gfCNCPoint2[7249] = {X 509.8909, Y 46.0603, Z -3.0000, A 0.000, B 0.000, C 0.000 }
gfCNCPoint2[7250] = {X 509.6596, Y 47.0980, Z -3.0000, A 0.000, B 0.000, C 0.000 }
gfCNCPoint2[7251] = {X 509.2797, Y 48.0910, Z -3.0000, A 0.000, B 0.000, C 0.000 }
gfCNCPoint2[7252] = {X 508.7593, Y 49.0180, Z -3.0000, A 0.000, B 0.000, C 0.000 }
gfCNCPoint2[7253] = {X 508.0200, Y 49.9571, Z -3.0000, A 0.000, B 0.000, C 0.000 }
gfCNCPoint2[7254] = {X 507.1371, Y 50.7626, Z -3.0000, A 0.000, B 0.000, C 0.000 }
gfCNCPoint2[7255] = {X 506.1343, Y 51.4129, Z -3.0000, A 0.000, B 0.000, C 0.000 }
gfCNCPoint2[7256] = {X 505.0386, Y 51.8902, Z -3.0000, A 0.000, B 0.000, C 0.000 }
gfCNCPoint2[7257] = {X 503.8796, Y 52.1819, Z -3.0000, A 0.000, B 0.000, C 0.000 }
gfCNCPoint2[7258] = {X 502.6885, Y 52.2800, Z -3.0000, A 0.000, B 0.000, C 0.000 }
gfCNCPoint2[7259] = {X 496.2450, Y 52.2800, Z -3.0000, A 0.000, B 0.000, C 0.000 }
gfCNCPoint2[7260] = {X 495.0845, Y 52.1869, Z -3.0000, A 0.000, B 0.000, C 0.000 }
gfCNCPoint2[7261] = {X 493.9538, Y 51.9100, Z -3.0000, A 0.000, B 0.000, C 0.000 }
gfCNCPoint2[7262] = {X 492.8816, Y 51.4564, Z -3.0000, A 0.000, B 0.000, C 0.000 }
gfCNCPoint2[7263] = {X 491.8954, Y 50.8377, Z -3.0000, A 0.000, B 0.000, C 0.000 }
gfCNCPoint2[7264] = {X 491.0204, Y 50.0697, Z -3.0000, A 0.000, B 0.000, C 0.000 }
gfCNCPoint2[7265] = {X 490.2980, Y 49.1989, Z -3.0000, A 0.000, B 0.000, C 0.000 }
gfCNCPoint2[7266] = {X 489.7192, Y 48.2267, Z -3.0000, A 0.000, B 0.000, C 0.000 }
gfCNCPoint2[7267] = {X 489.2980, Y 47.1766, Z -3.0000, A 0.000, B 0.000, C 0.000 }
gfCNCPoint2[7268] = {X 488.8769, Y 48.2267, Z -3.0000, A 0.000, B 0.000, C 0.000 }
gfCNCPoint2[7269] = {X 488.2981, Y 49.1989, Z -3.0000, A 0.000, B 0.000, C 0.000 }
gfCNCPoint2[7270] = {X 487.5756, Y 50.0697, Z -3.0000, A 0.000, B 0.000, C 0.000 }
gfCNCPoint2[7271] = {X 486.8824, Y 50.6978, Z -3.0000, A 0.000, B 0.000, C 0.000 }
gfCNCPoint2[7272] = {X 486.1145, Y 51.2318, Z -3.0000, A 0.000, B 0.000, C 0.000 }
gfCNCPoint2[7273] = {X 485.2843, Y 51.6629, Z -3.0000, A 0.000, B 0.000, C 0.000 }
gfCNCPoint2[7274] = {X 486.0586, Y 53.1385, Z -3.0000, A 0.000, B 0.000, C 0.000 }
gfCNCPoint2[7275] = {X 486.6224, Y 54.7067, Z -3.0000, A 0.000, B 0.000, C 0.000 }
gfCNCPoint2[7276] = {X 486.9651, Y 56.3375, Z -3.0000, A 0.000, B 0.000, C 0.000 }
gfCNCPoint2[7277] = {X 487.0800, Y 58.0000, Z -3.0000, A 0.000, B 0.000, C 0.000 }
gfCNCPoint2[7278] = {X 487.0796, Y 59.0339, Z -3.0000, A 0.000, B 0.000, C 0.000 }
gfCNCPoint2[7279] = {X 486.9596, Y 60.6353, Z -3.0000, A 0.000, B 0.000, C 0.000 }
gfCNCPoint2[7280] = {X 486.6283, Y 62.2067, Z -3.0000, A 0.000, B 0.000, C 0.000 }
gfCNCPoint2[7281] = {X 486.0914, Y 63.7202, Z -3.0000, A 0.000, B 0.000, C 0.000 }
gfCNCPoint2[7282] = {X 485.3585, Y 65.1491, Z -3.0000, A 0.000, B 0.000, C 0.000 }
gfCNCPoint2[7283] = {X 484.4426, Y 66.4682, Z -3.0000, A 0.000, B 0.000, C 0.000 }
gfCNCPoint2[7284] = {X 483.3598, Y 67.6542, Z -3.0000, A 0.000, B 0.000, C 0.000 }
gfCNCPoint2[7285] = {X 483.3601, Y 88.3509, Z -3.0000, A 0.000, B 0.000, C 0.000 }
gfCNCPoint2[7286] = {X 484.3099, Y 89.3715, Z -3.0000, A 0.000, B 0.000, C 0.000 }
gfCNCPoint2[7287] = {X 485.1356, Y 90.4950, Z -3.0000, A 0.000, B 0.000, C 0.000 }
gfCNCPoint2[7288] = {X 507.6818, Y 90.4950, Z -3.0000, A 0.000, B 0.000, C 0.000 }
gfCNCPoint2[7289] = {X 507.6818, Y 92.8950, Z -3.0000, A 0.000, B 0.000, C 0.000 }
gfCNCPoint2[7290] = {X 592.8965, Y 92.8950, Z -3.0000, A 0.000, B 0.000, C 0.000 }
gfCNCPoint2[7291] = {X 592.8965, Y 56.5812, Z -3.0000, A 0.000, B 0.000, C 0.000 }
gfCNCPoint2[7292] = {X 591.4810, Y 56.4128, Z -3.0000, A 0.000, B 0.000, C 0.000 }
gfCNCPoint2[7293] = {X 590.0968, Y 56.0720, Z -3.0000, A 0.000, B 0.000, C 0.000 }
gfCNCPoint2[7294] = {X 588.7648, Y 55.5641, Z -3.0000, A 0.000, B 0.000, C 0.000 }
gfCNCPoint2[7295] = {X 587.5052, Y 54.8965, Z -3.0000, A 0.000, B 0.000, C 0.000 }
gfCNCPoint2[7296] = {X 586.9690, Y 55.2051, Z -3.0000, A 0.000, B 0.000, C 0.000 }
gfCNCPoint2[7297] = {X 586.4171, Y 55.4846, Z -3.0000, A 0.000, B 0.000, C 0.000 }
gfCNCPoint2[7298] = {X 584.8782, Y 56.0830, Z -3.0000, A 0.000, B 0.000, C 0.000 }
gfCNCPoint2[7299] = {X 583.2699, Y 56.4570, Z -3.0000, A 0.000, B 0.000, C 0.000 }
gfCNCPoint2[7300] = {X 581.6248, Y 56.5987, Z -3.0000, A 0.000, B 0.000, C 0.000 }
gfCNCPoint2[7301] = {X 579.9763, Y 56.5055, Z -3.0000, A 0.000, B 0.000, C 0.000 }
gfCNCPoint2[7302] = {X 578.3577, Y 56.1792, Z -3.0000, A 0.000, B 0.000, C 0.000 }
gfCNCPoint2[7303] = {X 576.8018, Y 55.6263, Z -3.0000, A 0.000, B 0.000, C 0.000 }
gfCNCPoint2[7304] = {X 575.3401, Y 54.8581, Z -3.0000, A 0.000, B 0.000, C 0.000 }
gfCNCPoint2[7305] = {X 573.9176, Y 55.6091, Z -3.0000, A 0.000, B 0.000, C 0.000 }
gfCNCPoint2[7306] = {X 572.4049, Y 56.1560, Z -3.0000, A 0.000, B 0.000, C 0.000 }
gfCNCPoint2[7307] = {X 570.8311, Y 56.4885, Z -3.0000, A 0.000, B 0.000, C 0.000 }
gfCNCPoint2[7308] = {X 569.2264, Y 56.6000, Z -3.0000, A 0.000, B 0.000, C 0.000 }
gfCNCPoint2[7309] = {X 562.4443, Y 56.6000, Z -3.0000, A 0.000, B 0.000, C 0.000 }
gfCNCPoint2[7310] = {X 560.8792, Y 56.4939, Z -3.0000, A 0.000, B 0.000, C 0.000 }
gfCNCPoint2[7311] = {X 559.3428, Y 56.1777, Z -3.0000, A 0.000, B 0.000, C 0.000 }
gfCNCPoint2[7312] = {X 557.8630, Y 55.6570, Z -3.0000, A 0.000, B 0.000, C 0.000 }
gfCNCPoint2[7313] = {X 556.4671, Y 54.9415, Z -3.0000, A 0.000, B 0.000, C 0.000 }
gfCNCPoint2[7314] = {X 555.1804, Y 54.0441, Z -3.0000, A 0.000, B 0.000, C 0.000 }
gfCNCPoint2[7315] = {X 554.0266, Y 52.9814, Z -3.0000, A 0.000, B 0.000, C 0.000 }
gfCNCPoint2[7316] = {X 553.0267, Y 51.7727, Z -3.0000, A 0.000, B 0.000, C 0.000 }
gfCNCPoint2[7317] = {X 552.1991, Y 50.4401, Z -3.0000, A 0.000, B 0.000, C 0.000 }
gfCNCPoint2[7318] = {X 551.5587, Y 49.0081, Z -3.0000, A 0.000, B 0.000, C 0.000 }
gfCNCPoint2[7319] = {X 551.1637, Y 47.7032, Z -3.0000, A 0.000, B 0.000, C 0.000 }
gfCNCPoint2[7320] = {X 550.9244, Y 46.3610, Z -3.0000, A 0.000, B 0.000, C 0.000 }
gfCNCPoint2[7321] = {X 550.8443, Y 45.0000, Z -3.0000, A 0.000, B 0.000, C 0.000 }
gfCNCPoint2[7322] = {X 550.8443, Y 44.0535, Z -3.0000, A 0.000, B 0.000, C 0.000 }
gfCNCPoint2[7323] = {X 550.9571, Y 42.4679, Z -3.0000, A 0.000, B 0.000, C 0.000 }
gfCNCPoint2[7324] = {X 551.2850, Y 40.9124, Z -3.0000, A 0.000, B 0.000, C 0.000 }
gfCNCPoint2[7325] = {X 551.8218, Y 39.4161, Z -3.0000, A 0.000, B 0.000, C 0.000 }
gfCNCPoint2[7326] = {X 549.6234, Y 38.4533, Z -3.0000, A 0.000, B 0.000, C 0.000 }
gfCNCPoint2[7327] = {X 549.7925, Y 38.0819, Z -3.0000, A 0.000, B 0.000, C 0.000 }
gfCNCPoint2[7328] = {X 549.9724, Y 37.7156, Z -3.0000, A 0.000, B 0.000, C 0.000 }
gfCNCPoint2[7329] = {X 549.9724, Y 16.9500, Z -3.0000, A 0.000, B 0.000, C 0.000 }
gfCNCPoint2[7330] = {X 549.8029, Y 17.1990, Z -3.0000, A 0.000, B 0.000, C 0.000 }
gfCNCPoint2[7331] = {X 549.6232, Y 17.4407, Z -3.0000, A 0.000, B 0.000, C 0.000 }
gfCNCPoint2[7332] = {X 549.6234, Y 38.4533, Z -3.0000, A 0.000, B 0.000, C 0.000 }
gfCNCPoint2[7333] = {X 551.8218, Y 39.4161, Z -3.0000, A 0.000, B 0.000, C 0.000 }
gfCNCPoint2[7334] = {X 552.0826, Y 38.8609, Z -3.0000, A 0.000, B 0.000, C 0.000 }
gfCNCPoint2[7335] = {X 552.3724, Y 38.3202, Z -3.0000, A 0.000, B 0.000, C 0.000 }
gfCNCPoint2[7336] = {X 552.3724, Y 11.6888, Z -3.0000, A 0.000, B 0.000, C 0.000 }
gfCNCPoint2[7337] = {X 551.6708, Y 10.2343, Z -3.0000, A 0.000, B 0.000, C 0.000 }
gfCNCPoint2[7338] = {X 551.1780, Y 8.6964, Z -3.0000, A 0.000, B 0.000, C 0.000 }
gfCNCPoint2[7339] = {X 550.9035, Y 7.1050, Z -3.0000, A 0.000, B 0.000, C 0.000 }
gfCNCPoint2[7340] = {X 524.2928, Y 7.1050, Z -3.0000, A 0.000, B 0.000, C 0.000 }
gfCNCPoint2[7341] = {X 524.3789, Y 7.2067, Z -3.0000, A 0.000, B 0.000, C 0.000 }
gfCNCPoint2[7342] = {X 524.4621, Y 7.3107, Z -3.0000, A 0.000, B 0.000, C 0.000 }
gfCNCPoint2[7343] = {X 543.7426, Y 7.3112, Z -3.0000, A 0.000, B 0.000, C 0.000 }
gfCNCPoint2[7344] = {X 544.7118, Y 7.3834, Z -3.0000, A 0.000, B 0.000, C 0.000 }
gfCNCPoint2[7345] = {X 545.6475, Y 7.6459, Z -3.0000, A 0.000, B 0.000, C 0.000 }
gfCNCPoint2[7346] = {X 546.5127, Y 8.0885, Z -3.0000, A 0.000, B 0.000, C 0.000 }
gfCNCPoint2[7347] = {X 547.2732, Y 8.6936, Z -3.0000, A 0.000, B 0.000, C 0.000 }
gfCNCPoint2[7348] = {X 547.8989, Y 9.4373, Z -3.0000, A 0.000, B 0.000, C 0.000 }
gfCNCPoint2[7349] = {X 548.3649, Y 10.2901, Z -3.0000, A 0.000, B 0.000, C 0.000 }
gfCNCPoint2[7350] = {X 548.6529, Y 11.2183, Z -3.0000, A 0.000, B 0.000, C 0.000 }
gfCNCPoint2[7351] = {X 548.7514, Y 12.1852, Z -3.0000, A 0.000, B 0.000, C 0.000 }
gfCNCPoint2[7352] = {X 548.7512, Y 13.0283, Z -3.0000, A 0.000, B 0.000, C 0.000 }
gfCNCPoint2[7353] = {X 548.6549, Y 13.9439, Z -3.0000, A 0.000, B 0.000, C 0.000 }
gfCNCPoint2[7354] = {X 548.3884, Y 14.8251, Z -3.0000, A 0.000, B 0.000, C 0.000 }
gfCNCPoint2[7355] = {X 547.9611, Y 15.6406, Z -3.0000, A 0.000, B 0.000, C 0.000 }
gfCNCPoint2[7356] = {X 547.6183, Y 16.1045, Z -3.0000, A 0.000, B 0.000, C 0.000 }
gfCNCPoint2[7357] = {X 547.2232, Y 16.5248, Z -3.0000, A 0.000, B 0.000, C 0.000 }
gfCNCPoint2[7358] = {X 547.2234, Y 40.6622, Z -3.0000, A 0.000, B 0.000, C 0.000 }
gfCNCPoint2[7359] = {X 547.8650, Y 41.4042, Z -3.0000, A 0.000, B 0.000, C 0.000 }
gfCNCPoint2[7360] = {X 548.3452, Y 42.2595, Z -3.0000, A 0.000, B 0.000, C 0.000 }
gfCNCPoint2[7361] = {X 548.6447, Y 43.1936, Z -3.0000, A 0.000, B 0.000, C 0.000 }
gfCNCPoint2[7362] = {X 548.7513, Y 44.1687, Z -3.0000, A 0.000, B 0.000, C 0.000 }
gfCNCPoint2[7363] = {X 548.7514, Y 45.0016, Z -3.0000, A 0.000, B 0.000, C 0.000 }
gfCNCPoint2[7364] = {X 548.6696, Y 45.8828, Z -3.0000, A 0.000, B 0.000, C 0.000 }
gfCNCPoint2[7365] = {X 548.4300, Y 46.7348, Z -3.0000, A 0.000, B 0.000, C 0.000 }
gfCNCPoint2[7366] = {X 548.0407, Y 47.5296, Z -3.0000, A 0.000, B 0.000, C 0.000 }
gfCNCPoint2[7367] = {X 547.5144, Y 48.2411, Z -3.0000, A 0.000, B 0.000, C 0.000 }
gfCNCPoint2[7368] = {X 546.7288, Y 48.9506, Z -3.0000, A 0.000, B 0.000, C 0.000 }
gfCNCPoint2[7369] = {X 545.8088, Y 49.4742, Z -3.0000, A 0.000, B 0.000, C 0.000 }
gfCNCPoint2[7370] = {X 544.7975, Y 49.7874, Z -3.0000, A 0.000, B 0.000, C 0.000 }
gfCNCPoint2[7371] = {X 543.7426, Y 49.8753, Z -3.0000, A 0.000, B 0.000, C 0.000 }
gfCNCPoint2[7372] = {X 524.3233, Y 49.8758, Z -3.0000, A 0.000, B 0.000, C 0.000 }
gfCNCPoint2[7373] = {X 523.7105, Y 50.5147, Z -3.0000, A 0.000, B 0.000, C 0.000 }
gfCNCPoint2[7374] = {X 522.9953, Y 51.0365, Z -3.0000, A 0.000, B 0.000, C 0.000 }
gfCNCPoint2[7375] = {X 522.1999, Y 51.4251, Z -3.0000, A 0.000, B 0.000, C 0.000 }
gfCNCPoint2[7376] = {X 521.3487, Y 51.6685, Z -3.0000, A 0.000, B 0.000, C 0.000 }
gfCNCPoint2[7377] = {X 520.4681, Y 51.7591, Z -3.0000, A 0.000, B 0.000, C 0.000 }
gfCNCPoint2[7378] = {X 519.7998, Y 51.7591, Z -3.0000, A 0.000, B 0.000, C 0.000 }
gfCNCPoint2[7379] = {X 518.8477, Y 51.6654, Z -3.0000, A 0.000, B 0.000, C 0.000 }
gfCNCPoint2[7380] = {X 517.9323, Y 51.3877, Z -3.0000, A 0.000, B 0.000, C 0.000 }
gfCNCPoint2[7381] = {X 517.0886, Y 50.9367, Z -3.0000, A 0.000, B 0.000, C 0.000 }
gfCNCPoint2[7382] = {X 516.3491, Y 50.3298, Z -3.0000, A 0.000, B 0.000, C 0.000 }
gfCNCPoint2[7383] = {X 515.7422, Y 49.5903, Z -3.0000, A 0.000, B 0.000, C 0.000 }
gfCNCPoint2[7384] = {X 515.2912, Y 48.7466, Z -3.0000, A 0.000, B 0.000, C 0.000 }
gfCNCPoint2[7385] = {X 515.0135, Y 47.8312, Z -3.0000, A 0.000, B 0.000, C 0.000 }
gfCNCPoint2[7386] = {X 514.9198, Y 46.8791, Z -3.0000, A 0.000, B 0.000, C 0.000 }
gfCNCPoint2[7387] = {X 514.9198, Y 39.9011, Z -3.0000, A 0.000, B 0.000, C 0.000 }
gfCNCPoint2[7388] = {X 515.0197, Y 38.9186, Z -3.0000, A 0.000, B 0.000, C 0.000 }
gfCNCPoint2[7389] = {X 515.3154, Y 37.9764, Z -3.0000, A 0.000, B 0.000, C 0.000 }
gfCNCPoint2[7390] = {X 515.7947, Y 37.1129, Z -3.0000, A 0.000, B 0.000, C 0.000 }
gfCNCPoint2[7391] = {X 516.4381, Y 36.3637, Z -3.0000, A 0.000, B 0.000, C 0.000 }
gfCNCPoint2[7392] = {X 517.2191, Y 35.7593, Z -3.0000, A 0.000, B 0.000, C 0.000 }
gfCNCPoint2[7393] = {X 518.1058, Y 35.3245, Z -3.0000, A 0.000, B 0.000, C 0.000 }
gfCNCPoint2[7394] = {X 519.0619, Y 35.0772, Z -3.0000, A 0.000, B 0.000, C 0.000 }
gfCNCPoint2[7395] = {X 519.4084, Y 35.0368, Z -3.0000, A 0.000, B 0.000, C 0.000 }
gfCNCPoint2[7396] = {X 519.7568, Y 35.0213, Z -3.0000, A 0.000, B 0.000, C 0.000 }
gfCNCPoint2[7397] = {X 520.5345, Y 35.0216, Z -3.0000, A 0.000, B 0.000, C 0.000 }
gfCNCPoint2[7398] = {X 521.4086, Y 35.1126, Z -3.0000, A 0.000, B 0.000, C 0.000 }
gfCNCPoint2[7399] = {X 522.2522, Y 35.3589, Z -3.0000, A 0.000, B 0.000, C 0.000 }
gfCNCPoint2[7400] = {X 523.0379, Y 35.7525, Z -3.0000, A 0.000, B 0.000, C 0.000 }
gfCNCPoint2[7401] = {X 523.7403, Y 36.2806, Z -3.0000, A 0.000, B 0.000, C 0.000 }
gfCNCPoint2[7402] = {X 524.3366, Y 36.9262, Z -3.0000, A 0.000, B 0.000, C 0.000 }
gfCNCPoint2[7403] = {X 534.0719, Y 36.9267, Z -3.0000, A 0.000, B 0.000, C 0.000 }
gfCNCPoint2[7404] = {X 534.0719, Y 34.5249, Z -3.0000, A 0.000, B 0.000, C 0.000 }
gfCNCPoint2[7405] = {X 530.3966, Y 34.5246, Z -3.0000, A 0.000, B 0.000, C 0.000 }
gfCNCPoint2[7406] = {X 529.7967, Y 35.1733, Z -3.0000, A 0.000, B 0.000, C 0.000 }
gfCNCPoint2[7407] = {X 529.0897, Y 35.7033, Z -3.0000, A 0.000, B 0.000, C 0.000 }
gfCNCPoint2[7408] = {X 528.2986, Y 36.0971, Z -3.0000, A 0.000, B 0.000, C 0.000 }
gfCNCPoint2[7409] = {X 527.4495, Y 36.3417, Z -3.0000, A 0.000, B 0.000, C 0.000 }
gfCNCPoint2[7410] = {X 526.5703, Y 36.4293, Z -3.0000, A 0.000, B 0.000, C 0.000 }
gfCNCPoint2[7411] = {X 525.8868, Y 36.4294, Z -3.0000, A 0.000, B 0.000, C 0.000 }
gfCNCPoint2[7412] = {X 524.9094, Y 36.3306, Z -3.0000, A 0.000, B 0.000, C 0.000 }
gfCNCPoint2[7413] = {X 523.9717, Y 36.0380, Z -3.0000, A 0.000, B 0.000, C 0.000 }
gfCNCPoint2[7414] = {X 523.1116, Y 35.5636, Z -3.0000, A 0.000, B 0.000, C 0.000 }
gfCNCPoint2[7415] = {X 522.3639, Y 34.9265, Z -3.0000, A 0.000, B 0.000, C 0.000 }
gfCNCPoint2[7416] = {X 521.7590, Y 34.1525, Z -3.0000, A 0.000, B 0.000, C 0.000 }
gfCNCPoint2[7417] = {X 521.3213, Y 33.2731, Z -3.0000, A 0.000, B 0.000, C 0.000 }
gfCNCPoint2[7418] = {X 521.0686, Y 32.3239, Z -3.0000, A 0.000, B 0.000, C 0.000 }
gfCNCPoint2[7419] = {X 521.0222, Y 31.9379, Z -3.0000, A 0.000, B 0.000, C 0.000 }
gfCNCPoint2[7420] = {X 521.0068, Y 31.5495, Z -3.0000, A 0.000, B 0.000, C 0.000 }
gfCNCPoint2[7421] = {X 521.0076, Y 24.4815, Z -3.0000, A 0.000, B 0.000, C 0.000 }
gfCNCPoint2[7422] = {X 521.0984, Y 23.6300, Z -3.0000, A 0.000, B 0.000, C 0.000 }
gfCNCPoint2[7423] = {X 521.3368, Y 22.8074, Z -3.0000, A 0.000, B 0.000, C 0.000 }
gfCNCPoint2[7424] = {X 521.7152, Y 22.0391, Z -3.0000, A 0.000, B 0.000, C 0.000 }
gfCNCPoint2[7425] = {X 521.1864, Y 22.1316, Z -3.0000, A 0.000, B 0.000, C 0.000 }
gfCNCPoint2[7426] = {X 520.6505, Y 22.1656, Z -3.0000, A 0.000, B 0.000, C 0.000 }
gfCNCPoint2[7427] = {X 519.9691, Y 22.1657, Z -3.0000, A 0.000, B 0.000, C 0.000 }
gfCNCPoint2[7428] = {X 519.5109, Y 22.1442, Z -3.0000, A 0.000, B 0.000, C 0.000 }
gfCNCPoint2[7429] = {X 519.0567, Y 22.0797, Z -3.0000, A 0.000, B 0.000, C 0.000 }
gfCNCPoint2[7430] = {X 518.1336, Y 21.8074, Z -3.0000, A 0.000, B 0.000, C 0.000 }
gfCNCPoint2[7431] = {X 517.2820, Y 21.3592, Z -3.0000, A 0.000, B 0.000, C 0.000 }
gfCNCPoint2[7432] = {X 516.5348, Y 20.7527, Z -3.0000, A 0.000, B 0.000, C 0.000 }
gfCNCPoint2[7433] = {X 515.9212, Y 20.0113, Z -3.0000, A 0.000, B 0.000, C 0.000 }
gfCNCPoint2[7434] = {X 515.4650, Y 19.1639, Z -3.0000, A 0.000, B 0.000, C 0.000 }
gfCNCPoint2[7435] = {X 515.1840, Y 18.2434, Z -3.0000, A 0.000, B 0.000, C 0.000 }
gfCNCPoint2[7436] = {X 515.0891, Y 17.2857, Z -3.0000, A 0.000, B 0.000, C 0.000 }
gfCNCPoint2[7437] = {X 515.0891, Y 10.3077, Z -3.0000, A 0.000, B 0.000, C 0.000 }
gfCNCPoint2[7438] = {X 515.0965, Y 10.0383, Z -3.0000, A 0.000, B 0.000, C 0.000 }
gfCNCPoint2[7439] = {X 515.1189, Y 9.7697, Z -3.0000, A 0.000, B 0.000, C 0.000 }
gfCNCPoint2[7440] = {X 515.3251, Y 8.8084, Z -3.0000, A 0.000, B 0.000, C 0.000 }
gfCNCPoint2[7441] = {X 515.7199, Y 7.9080, Z -3.0000, A 0.000, B 0.000, C 0.000 }
gfCNCPoint2[7442] = {X 516.2871, Y 7.1050, Z -3.0000, A 0.000, B 0.000, C 0.000 }
gfCNCPoint2[7443] = {X 516.6492, Y 7.4201, Z -3.0000, A 0.000, B 0.000, C 0.000 }
gfCNCPoint2[7444] = {X 517.3373, Y 6.7816, Z -3.0000, A 0.000, B 0.000, C 0.000 }
gfCNCPoint2[7445] = {X 518.1451, Y 6.3036, Z -3.0000, A 0.000, B 0.000, C 0.000 }
gfCNCPoint2[7446] = {X 519.0359, Y 6.0078, Z -3.0000, A 0.000, B 0.000, C 0.000 }
gfCNCPoint2[7447] = {X 519.9692, Y 5.9077, Z -3.0000, A 0.000, B 0.000, C 0.000 }
gfCNCPoint2[7448] = {X 520.6509, Y 5.9079, Z -3.0000, A 0.000, B 0.000, C 0.000 }
gfCNCPoint2[7449] = {X 521.4834, Y 5.9951, Z -3.0000, A 0.000, B 0.000, C 0.000 }
gfCNCPoint2[7450] = {X 522.2844, Y 6.2384, Z -3.0000, A 0.000, B 0.000, C 0.000 }
gfCNCPoint2[7451] = {X 523.0248, Y 6.6290, Z -3.0000, A 0.000, B 0.000, C 0.000 }
gfCNCPoint2[7452] = {X 523.6778, Y 7.1528, Z -3.0000, A 0.000, B 0.000, C 0.000 }
gfCNCPoint2[7453] = {X 524.2198, Y 7.7907, Z -3.0000, A 0.000, B 0.000, C 0.000 }
gfCNCPoint2[7454] = {X 543.7489, Y 7.7912, Z -3.0000, A 0.000, B 0.000, C 0.000 }
gfCNCPoint2[7455] = {X 544.7470, Y 7.8786, Z -3.0000, A 0.000, B 0.000, C 0.000 }
gfCNCPoint2[7456] = {X 545.6995, Y 8.1892, Z -3.0000, A 0.000, B 0.000, C 0.000 }
gfCNCPoint2[7457] = {X 546.5572, Y 8.7070, Z -3.0000, A 0.000, B 0.000, C 0.000 }
gfCNCPoint2[7458] = {X 547.2757, Y 9.4052, Z -3.0000, A 0.000, B 0.000, C 0.000 }
gfCNCPoint2[7459] = {X 547.8178, Y 10.2477, Z -3.0000, A 0.000, B 0.000, C 0.000 }
gfCNCPoint2[7460] = {X 548.1556, Y 11.1909, Z -3.0000, A 0.000, B 0.000, C 0.000 }
gfCNCPoint2[7461] = {X 548.2714, Y 12.1861, Z -3.0000, A 0.000, B 0.000, C 0.000 }
gfCNCPoint2[7462] = {X 548.2712, Y 13.0233, Z -3.0000, A 0.000, B 0.000, C 0.000 }
gfCNCPoint2[7463] = {X 548.1628, Y 13.9496, Z -3.0000, A 0.000, B 0.000, C 0.000 }
gfCNCPoint2[7464] = {X 547.8617, Y 14.8322, Z -3.0000, A 0.000, B 0.000, C 0.000 }
gfCNCPoint2[7465] = {X 547.3813, Y 15.6315, Z -3.0000, A 0.000, B 0.000, C 0.000 }
gfCNCPoint2[7466] = {X 546.7432, Y 16.3116, Z -3.0000, A 0.000, B 0.000, C 0.000 }
gfCNCPoint2[7467] = {X 546.7434, Y 40.8754, Z -3.0000, A 0.000, B 0.000, C 0.000 }
gfCNCPoint2[7468] = {X 547.3883, Y 41.5646, Z -3.0000, A 0.000, B 0.000, C 0.000 }
gfCNCPoint2[7469] = {X 547.8713, Y 42.3754, Z -3.0000, A 0.000, B 0.000, C 0.000 }
gfCNCPoint2[7470] = {X 548.1702, Y 43.2706, Z -3.0000, A 0.000, B 0.000, C 0.000 }
gfCNCPoint2[7471] = {X 548.2714, Y 44.2089, Z -3.0000, A 0.000, B 0.000, C 0.000 }
gfCNCPoint2[7472] = {X 548.2714, Y 45.0007, Z -3.0000, A 0.000, B 0.000, C 0.000 }
gfCNCPoint2[7473] = {X 548.1556, Y 45.9959, Z -3.0000, A 0.000, B 0.000, C 0.000 }
gfCNCPoint2[7474] = {X 547.8178, Y 46.9391, Z -3.0000, A 0.000, B 0.000, C 0.000 }
gfCNCPoint2[7475] = {X 547.2757, Y 47.7816, Z -3.0000, A 0.000, B 0.000, C 0.000 }
gfCNCPoint2[7476] = {X 546.5572, Y 48.4798, Z -3.0000, A 0.000, B 0.000, C 0.000 }
gfCNCPoint2[7477] = {X 545.6995, Y 48.9975, Z -3.0000, A 0.000, B 0.000, C 0.000 }
gfCNCPoint2[7478] = {X 544.7469, Y 49.3080, Z -3.0000, A 0.000, B 0.000, C 0.000 }
gfCNCPoint2[7479] = {X 543.7489, Y 49.3953, Z -3.0000, A 0.000, B 0.000, C 0.000 }
gfCNCPoint2[7480] = {X 524.0859, Y 49.3958, Z -3.0000, A 0.000, B 0.000, C 0.000 }
gfCNCPoint2[7481] = {X 523.5292, Y 50.0308, Z -3.0000, A 0.000, B 0.000, C 0.000 }
gfCNCPoint2[7482] = {X 522.8649, Y 50.5523, Z -3.0000, A 0.000, B 0.000, C 0.000 }
gfCNCPoint2[7483] = {X 522.1158, Y 50.9422, Z -3.0000, A 0.000, B 0.000, C 0.000 }
gfCNCPoint2[7484] = {X 521.3076, Y 51.1873, Z -3.0000, A 0.000, B 0.000, C 0.000 }
gfCNCPoint2[7485] = {X 520.4681, Y 51.2791, Z -3.0000, A 0.000, B 0.000, C 0.000 }
gfCNCPoint2[7486] = {X 519.7998, Y 51.2791, Z -3.0000, A 0.000, B 0.000, C 0.000 }
gfCNCPoint2[7487] = {X 518.8207, Y 51.1688, Z -3.0000, A 0.000, B 0.000, C 0.000 }
gfCNCPoint2[7488] = {X 517.8907, Y 50.8434, Z -3.0000, A 0.000, B 0.000, C 0.000 }
gfCNCPoint2[7489] = {X 517.0564, Y 50.3192, Z -3.0000, A 0.000, B 0.000, C 0.000 }
gfCNCPoint2[7490] = {X 516.3597, Y 49.6225, Z -3.0000, A 0.000, B 0.000, C 0.000 }
gfCNCPoint2[7491] = {X 515.8355, Y 48.7882, Z -3.0000, A 0.000, B 0.000, C 0.000 }
gfCNCPoint2[7492] = {X 515.5101, Y 47.8582, Z -3.0000, A 0.000, B 0.000, C 0.000 }
gfCNCPoint2[7493] = {X 515.3998, Y 46.8791, Z -3.0000, A 0.000, B 0.000, C 0.000 }
gfCNCPoint2[7494] = {X 515.3998, Y 39.9011, Z -3.0000, A 0.000, B 0.000, C 0.000 }
gfCNCPoint2[7495] = {X 515.5101, Y 38.9220, Z -3.0000, A 0.000, B 0.000, C 0.000 }
gfCNCPoint2[7496] = {X 515.8355, Y 37.9920, Z -3.0000, A 0.000, B 0.000, C 0.000 }
gfCNCPoint2[7497] = {X 516.3597, Y 37.1577, Z -3.0000, A 0.000, B 0.000, C 0.000 }
gfCNCPoint2[7498] = {X 517.0565, Y 36.4610, Z -3.0000, A 0.000, B 0.000, C 0.000 }
gfCNCPoint2[7499] = {X 517.8907, Y 35.9368, Z -3.0000, A 0.000, B 0.000, C 0.000 }
gfCNCPoint2[7500] = {X 518.8207, Y 35.6114, Z -3.0000, A 0.000, B 0.000, C 0.000 }
gfCNCPoint2[7501] = {X 519.7999, Y 35.5011, Z -3.0000, A 0.000, B 0.000, C 0.000 }
gfCNCPoint2[7502] = {X 520.5280, Y 35.5015, Z -3.0000, A 0.000, B 0.000, C 0.000 }
gfCNCPoint2[7503] = {X 521.3615, Y 35.5927, Z -3.0000, A 0.000, B 0.000, C 0.000 }
gfCNCPoint2[7504] = {X 522.1626, Y 35.8404, Z -3.0000, A 0.000, B 0.000, C 0.000 }
gfCNCPoint2[7505] = {X 522.9022, Y 36.2356, Z -3.0000, A 0.000, B 0.000, C 0.000 }
gfCNCPoint2[7506] = {X 523.5534, Y 36.7640, Z -3.0000, A 0.000, B 0.000, C 0.000 }
gfCNCPoint2[7507] = {X 524.0925, Y 37.4062, Z -3.0000, A 0.000, B 0.000, C 0.000 }
gfCNCPoint2[7508] = {X 534.5519, Y 37.4067, Z -3.0000, A 0.000, B 0.000, C 0.000 }
gfCNCPoint2[7509] = {X 534.5519, Y 34.0450, Z -3.0000, A 0.000, B 0.000, C 0.000 }
gfCNCPoint2[7510] = {X 530.1526, Y 34.0445, Z -3.0000, A 0.000, B 0.000, C 0.000 }
gfCNCPoint2[7511] = {X 529.6049, Y 34.6951, Z -3.0000, A 0.000, B 0.000, C 0.000 }
gfCNCPoint2[7512] = {X 528.9423, Y 35.2282, Z -3.0000, A 0.000, B 0.000, C 0.000 }
gfCNCPoint2[7513] = {X 528.1895, Y 35.6238, Z -3.0000, A 0.000, B 0.000, C 0.000 }
gfCNCPoint2[7514] = {X 527.3747, Y 35.8673, Z -3.0000, A 0.000, B 0.000, C 0.000 }
gfCNCPoint2[7515] = {X 526.5283, Y 35.9495, Z -3.0000, A 0.000, B 0.000, C 0.000 }
gfCNCPoint2[7516] = {X 525.8868, Y 35.9495, Z -3.0000, A 0.000, B 0.000, C 0.000 }
gfCNCPoint2[7517] = {X 524.9077, Y 35.8391, Z -3.0000, A 0.000, B 0.000, C 0.000 }
gfCNCPoint2[7518] = {X 523.9777, Y 35.5137, Z -3.0000, A 0.000, B 0.000, C 0.000 }
gfCNCPoint2[7519] = {X 523.1434, Y 34.9895, Z -3.0000, A 0.000, B 0.000, C 0.000 }
gfCNCPoint2[7520] = {X 522.4467, Y 34.2928, Z -3.0000, A 0.000, B 0.000, C 0.000 }
gfCNCPoint2[7521] = {X 521.9225, Y 33.4585, Z -3.0000, A 0.000, B 0.000, C 0.000 }
gfCNCPoint2[7522] = {X 521.5971, Y 32.5285, Z -3.0000, A 0.000, B 0.000, C 0.000 }
gfCNCPoint2[7523] = {X 521.4868, Y 31.5495, Z -3.0000, A 0.000, B 0.000, C 0.000 }
gfCNCPoint2[7524] = {X 521.4868, Y 24.5714, Z -3.0000, A 0.000, B 0.000, C 0.000 }
gfCNCPoint2[7525] = {X 521.5971, Y 23.5923, Z -3.0000, A 0.000, B 0.000, C 0.000 }
gfCNCPoint2[7526] = {X 521.9225, Y 22.6623, Z -3.0000, A 0.000, B 0.000, C 0.000 }
gfCNCPoint2[7527] = {X 522.4467, Y 21.8281, Z -3.0000, A 0.000, B 0.000, C 0.000 }
gfCNCPoint2[7528] = {X 523.1434, Y 21.1314, Z -3.0000, A 0.000, B 0.000, C 0.000 }
gfCNCPoint2[7529] = {X 523.9777, Y 20.6072, Z -3.0000, A 0.000, B 0.000, C 0.000 }
gfCNCPoint2[7530] = {X 524.9077, Y 20.2817, Z -3.0000, A 0.000, B 0.000, C 0.000 }
gfCNCPoint2[7531] = {X 525.8868, Y 20.1714, Z -3.0000, A 0.000, B 0.000, C 0.000 }
gfCNCPoint2[7532] = {X 526.5702, Y 20.1716, Z -3.0000, A 0.000, B 0.000, C 0.000 }
gfCNCPoint2[7533] = {X 527.4024, Y 20.2591, Z -3.0000, A 0.000, B 0.000, C 0.000 }
gfCNCPoint2[7534] = {X 528.2030, Y 20.5025, Z -3.0000, A 0.000, B 0.000, C 0.000 }
gfCNCPoint2[7535] = {X 528.9430, Y 20.8931, Z -3.0000, A 0.000, B 0.000, C 0.000 }
gfCNCPoint2[7536] = {X 529.5956, Y 21.4167, Z -3.0000, A 0.000, B 0.000, C 0.000 }
gfCNCPoint2[7537] = {X 530.1374, Y 22.0544, Z -3.0000, A 0.000, B 0.000, C 0.000 }
gfCNCPoint2[7538] = {X 534.5519, Y 22.0547, Z -3.0000, A 0.000, B 0.000, C 0.000 }
gfCNCPoint2[7539] = {X 534.5519, Y 19.7814, Z -3.0000, A 0.000, B 0.000, C 0.000 }
gfCNCPoint2[7540] = {X 528.8167, Y 19.7812, Z -3.0000, A 0.000, B 0.000, C 0.000 }
gfCNCPoint2[7541] = {X 528.8167, Y 20.2612, Z -3.0000, A 0.000, B 0.000, C 0.000 }
gfCNCPoint2[7542] = {X 534.0719, Y 20.2614, Z -3.0000, A 0.000, B 0.000, C 0.000 }
gfCNCPoint2[7543] = {X 534.0719, Y 21.5747, Z -3.0000, A 0.000, B 0.000, C 0.000 }
gfCNCPoint2[7544] = {X 530.3797, Y 21.5744, Z -3.0000, A 0.000, B 0.000, C 0.000 }
gfCNCPoint2[7545] = {X 529.6676, Y 20.8352, Z -3.0000, A 0.000, B 0.000, C 0.000 }
gfCNCPoint2[7546] = {X 528.8167, Y 20.2612, Z -3.0000, A 0.000, B 0.000, C 0.000 }
gfCNCPoint2[7547] = {X 528.8167, Y 19.7812, Z -3.0000, A 0.000, B 0.000, C 0.000 }
gfCNCPoint2[7548] = {X 524.2348, Y 19.7810, Z -3.0000, A 0.000, B 0.000, C 0.000 }
gfCNCPoint2[7549] = {X 523.6871, Y 20.4315, Z -3.0000, A 0.000, B 0.000, C 0.000 }
gfCNCPoint2[7550] = {X 523.0246, Y 20.9645, Z -3.0000, A 0.000, B 0.000, C 0.000 }
gfCNCPoint2[7551] = {X 522.2718, Y 21.3601, Z -3.0000, A 0.000, B 0.000, C 0.000 }
gfCNCPoint2[7552] = {X 521.4571, Y 21.6036, Z -3.0000, A 0.000, B 0.000, C 0.000 }
gfCNCPoint2[7553] = {X 520.6107, Y 21.6857, Z -3.0000, A 0.000, B 0.000, C 0.000 }
gfCNCPoint2[7554] = {X 519.9691, Y 21.6857, Z -3.0000, A 0.000, B 0.000, C 0.000 }
gfCNCPoint2[7555] = {X 518.9900, Y 21.5754, Z -3.0000, A 0.000, B 0.000, C 0.000 }
gfCNCPoint2[7556] = {X 518.0600, Y 21.2500, Z -3.0000, A 0.000, B 0.000, C 0.000 }
gfCNCPoint2[7557] = {X 517.2257, Y 20.7258, Z -3.0000, A 0.000, B 0.000, C 0.000 }
gfCNCPoint2[7558] = {X 516.5290, Y 20.0291, Z -3.0000, A 0.000, B 0.000, C 0.000 }
gfCNCPoint2[7559] = {X 516.0048, Y 19.1948, Z -3.0000, A 0.000, B 0.000, C 0.000 }
gfCNCPoint2[7560] = {X 515.6794, Y 18.2648, Z -3.0000, A 0.000, B 0.000, C 0.000 }
gfCNCPoint2[7561] = {X 515.5691, Y 17.2857, Z -3.0000, A 0.000, B 0.000, C 0.000 }
gfCNCPoint2[7562] = {X 515.5691, Y 10.3077, Z -3.0000, A 0.000, B 0.000, C 0.000 }
gfCNCPoint2[7563] = {X 515.6394, Y 9.5244, Z -3.0000, A 0.000, B 0.000, C 0.000 }
gfCNCPoint2[7564] = {X 515.8480, Y 8.7662, Z -3.0000, A 0.000, B 0.000, C 0.000 }
gfCNCPoint2[7565] = {X 516.1882, Y 8.0572, Z -3.0000, A 0.000, B 0.000, C 0.000 }
gfCNCPoint2[7566] = {X 516.6492, Y 7.4201, Z -3.0000, A 0.000, B 0.000, C 0.000 }
gfCNCPoint2[7567] = {X 516.2871, Y 7.1050, Z -3.0000, A 0.000, B 0.000, C 0.000 }
gfCNCPoint2[7568] = {X 469.2610, Y 7.1050, Z -3.0000, A 0.000, B 0.000, C 0.000 }
gfCNCPoint2[7569] = {X 469.2610, Y 11.9050, Z -3.0000, A 0.000, B 0.000, C 0.000 }
gfCNCPoint2[7570] = {X 469.1140, Y 11.9050, Z -3.0000, A 0.000, B 0.000, C 0.000 }
gfCNCPoint2[7571] = {X 469.1169, Y 12.0441, Z -3.0000, A 0.000, B 0.000, C 0.000 }
gfCNCPoint2[7572] = {X 469.1179, Y 12.1832, Z -3.0000, A 0.000, B 0.000, C 0.000 }
gfCNCPoint2[7573] = {X 469.1888, Y 12.0438, Z -3.0000, A 0.000, B 0.000, C 0.000 }
gfCNCPoint2[7574] = {X 469.2610, Y 11.9050, Z -3.0000, A 0.000, B 0.000, C 0.000 }
gfCNCPoint2[7575] = {X 469.2610, Y 9.5050, Z -3.0000, A 0.000, B 0.000, C 0.000 }
gfCNCPoint2[7576] = {X 466.2070, Y 9.5050, Z -3.0000, A 0.000, B 0.000, C 0.000 }
gfCNCPoint2[7577] = {X 466.5688, Y 10.7173, Z -3.0000, A 0.000, B 0.000, C 0.000 }
gfCNCPoint2[7578] = {X 466.7149, Y 11.9739, Z -3.0000, A 0.000, B 0.000, C 0.000 }
gfCNCPoint2[7579] = {X 466.7172, Y 12.0782, Z -3.0000, A 0.000, B 0.000, C 0.000 }
gfCNCPoint2[7580] = {X 466.7179, Y 12.1826, Z -3.0000, A 0.000, B 0.000, C 0.000 }
gfCNCPoint2[7581] = {X 466.7179, Y 12.9779, Z -3.0000, A 0.000, B 0.000, C 0.000 }
gfCNCPoint2[7582] = {X 466.6191, Y 14.1736, Z -3.0000, A 0.000, B 0.000, C 0.000 }
gfCNCPoint2[7583] = {X 466.3252, Y 15.3368, Z -3.0000, A 0.000, B 0.000, C 0.000 }
gfCNCPoint2[7584] = {X 465.8443, Y 16.4359, Z -3.0000, A 0.000, B 0.000, C 0.000 }
gfCNCPoint2[7585] = {X 465.1893, Y 17.4412, Z -3.0000, A 0.000, B 0.000, C 0.000 }
gfCNCPoint2[7586] = {X 465.1897, Y 25.8716, Z -3.0000, A 0.000, B 0.000, C 0.000 }
gfCNCPoint2[7587] = {X 467.5897, Y 25.8714, Z -3.0000, A 0.000, B 0.000, C 0.000 }
gfCNCPoint2[7588] = {X 467.5904, Y 38.9895, Z -3.0000, A 0.000, B 0.000, C 0.000 }
gfCNCPoint2[7589] = {X 467.6015, Y 39.0069, Z -3.0000, A 0.000, B 0.000, C 0.000 }
gfCNCPoint2[7590] = {X 468.3506, Y 37.9855, Z -3.0000, A 0.000, B 0.000, C 0.000 }
gfCNCPoint2[7591] = {X 469.2267, Y 37.0706, Z -3.0000, A 0.000, B 0.000, C 0.000 }
gfCNCPoint2[7592] = {X 470.2148, Y 36.2780, Z -3.0000, A 0.000, B 0.000, C 0.000 }
gfCNCPoint2[7593] = {X 471.5280, Y 33.7075, Z -3.0000, A 0.000, B 0.000, C 0.000 }
gfCNCPoint2[7594] = {X 470.4811, Y 32.4115, Z -3.0000, A 0.000, B 0.000, C 0.000 }
gfCNCPoint2[7595] = {X 469.5675, Y 31.0183, Z -3.0000, A 0.000, B 0.000, C 0.000 }
gfCNCPoint2[7596] = {X 468.7961, Y 29.5416, Z -3.0000, A 0.000, B 0.000, C 0.000 }
gfCNCPoint2[7597] = {X 468.1745, Y 27.9959, Z -3.0000, A 0.000, B 0.000, C 0.000 }
gfCNCPoint2[7598] = {X 467.7088, Y 26.3963, Z -3.0000, A 0.000, B 0.000, C 0.000 }
gfCNCPoint2[7599] = {X 467.6476, Y 26.1342, Z -3.0000, A 0.000, B 0.000, C 0.000 }
gfCNCPoint2[7600] = {X 467.5897, Y 25.8714, Z -3.0000, A 0.000, B 0.000, C 0.000 }
gfCNCPoint2[7601] = {X 465.1897, Y 25.8716, Z -3.0000, A 0.000, B 0.000, C 0.000 }
gfCNCPoint2[7602] = {X 465.1904, Y 39.7470, Z -3.0000, A 0.000, B 0.000, C 0.000 }
gfCNCPoint2[7603] = {X 465.3903, Y 40.0173, Z -3.0000, A 0.000, B 0.000, C 0.000 }
gfCNCPoint2[7604] = {X 465.5774, Y 40.2966, Z -3.0000, A 0.000, B 0.000, C 0.000 }
gfCNCPoint2[7605] = {X 466.0634, Y 41.1919, Z -3.0000, A 0.000, B 0.000, C 0.000 }
gfCNCPoint2[7606] = {X 466.4196, Y 42.1462, Z -3.0000, A 0.000, B 0.000, C 0.000 }
gfCNCPoint2[7607] = {X 466.6392, Y 43.1408, Z -3.0000, A 0.000, B 0.000, C 0.000 }
gfCNCPoint2[7608] = {X 466.7178, Y 44.1564, Z -3.0000, A 0.000, B 0.000, C 0.000 }
gfCNCPoint2[7609] = {X 466.7179, Y 45.0000, Z -3.0000, A 0.000, B 0.000, C 0.000 }
gfCNCPoint2[7610] = {X 466.7033, Y 45.4609, Z -3.0000, A 0.000, B 0.000, C 0.000 }
gfCNCPoint2[7611] = {X 466.6596, Y 45.9200, Z -3.0000, A 0.000, B 0.000, C 0.000 }
gfCNCPoint2[7612] = {X 468.5433, Y 45.9200, Z -3.0000, A 0.000, B 0.000, C 0.000 }
gfCNCPoint2[7613] = {X 468.4996, Y 45.4609, Z -3.0000, A 0.000, B 0.000, C 0.000 }
gfCNCPoint2[7614] = {X 468.4850, Y 45.0000, Z -3.0000, A 0.000, B 0.000, C 0.000 }
gfCNCPoint2[7615] = {X 468.4850, Y 44.2090, Z -3.0000, A 0.000, B 0.000, C 0.000 }
gfCNCPoint2[7616] = {X 468.5580, Y 43.1798, Z -3.0000, A 0.000, B 0.000, C 0.000 }
gfCNCPoint2[7617] = {X 468.7759, Y 42.1714, Z -3.0000, A 0.000, B 0.000, C 0.000 }
gfCNCPoint2[7618] = {X 469.1341, Y 41.2038, Z -3.0000, A 0.000, B 0.000, C 0.000 }
gfCNCPoint2[7619] = {X 469.6255, Y 40.2966, Z -3.0000, A 0.000, B 0.000, C 0.000 }
gfCNCPoint2[7620] = {X 470.3102, Y 39.3876, Z -3.0000, A 0.000, B 0.000, C 0.000 }
gfCNCPoint2[7621] = {X 471.1282, Y 38.5964, Z -3.0000, A 0.000, B 0.000, C 0.000 }
gfCNCPoint2[7622] = {X 472.0595, Y 37.9424, Z -3.0000, A 0.000, B 0.000, C 0.000 }
gfCNCPoint2[7623] = {X 474.4571, Y 33.2493, Z -3.0000, A 0.000, B 0.000, C 0.000 }
gfCNCPoint2[7624] = {X 473.2258, Y 32.0046, Z -3.0000, A 0.000, B 0.000, C 0.000 }
gfCNCPoint2[7625] = {X 472.1543, Y 30.6200, Z -3.0000, A 0.000, B 0.000, C 0.000 }
gfCNCPoint2[7626] = {X 471.2583, Y 29.1158, Z -3.0000, A 0.000, B 0.000, C 0.000 }
gfCNCPoint2[7627] = {X 470.5511, Y 27.5141, Z -3.0000, A 0.000, B 0.000, C 0.000 }
gfCNCPoint2[7628] = {X 470.0431, Y 25.8386, Z -3.0000, A 0.000, B 0.000, C 0.000 }
gfCNCPoint2[7629] = {X 469.9884, Y 25.6042, Z -3.0000, A 0.000, B 0.000, C 0.000 }
gfCNCPoint2[7630] = {X 469.9366, Y 25.3692, Z -3.0000, A 0.000, B 0.000, C 0.000 }
gfCNCPoint2[7631] = {X 469.6270, Y 23.4764, Z -3.0000, A 0.000, B 0.000, C 0.000 }
gfCNCPoint2[7632] = {X 469.5028, Y 21.5625, Z -3.0000, A 0.000, B 0.000, C 0.000 }
gfCNCPoint2[7633] = {X 469.5652, Y 19.6455, Z -3.0000, A 0.000, B 0.000, C 0.000 }
gfCNCPoint2[7634] = {X 469.8136, Y 17.7437, Z -3.0000, A 0.000, B 0.000, C 0.000 }
gfCNCPoint2[7635] = {X 470.2458, Y 15.8751, Z -3.0000, A 0.000, B 0.000, C 0.000 }
gfCNCPoint2[7636] = {X 470.6919, Y 14.5440, Z -3.0000, A 0.000, B 0.000, C 0.000 }
gfCNCPoint2[7637] = {X 471.2622, Y 13.2612, Z -3.0000, A 0.000, B 0.000, C 0.000 }
gfCNCPoint2[7638] = {X 471.3232, Y 13.1413, Z -3.0000, A 0.000, B 0.000, C 0.000 }
gfCNCPoint2[7639] = {X 471.3853, Y 13.0219, Z -3.0000, A 0.000, B 0.000, C 0.000 }
gfCNCPoint2[7640] = {X 472.1263, Y 11.7667, Z -3.0000, A 0.000, B 0.000, C 0.000 }
gfCNCPoint2[7641] = {X 472.9873, Y 10.5907, Z -3.0000, A 0.000, B 0.000, C 0.000 }
gfCNCPoint2[7642] = {X 473.9599, Y 9.5050, Z -3.0000, A 0.000, B 0.000, C 0.000 }
gfCNCPoint2[7643] = {X 469.2610, Y 9.5050, Z -3.0000, A 0.000, B 0.000, C 0.000 }
gfCNCPoint2[7644] = {X 469.2610, Y 7.1050, Z -3.0000, A 0.000, B 0.000, C 0.000 }
gfCNCPoint2[7645] = {X 370.1021, Y 7.1050, Z -3.0000, A 0.000, B 0.000, C 0.000 }
gfCNCPoint2[7646] = {X 371.1257, Y 8.7920, Z -3.0000, A 0.000, B 0.000, C 0.000 }
gfCNCPoint2[7647] = {X 372.0365, Y 10.5424, Z -3.0000, A 0.000, B 0.000, C 0.000 }
gfCNCPoint2[7648] = {X 372.9307, Y 12.6018, Z -3.0000, A 0.000, B 0.000, C 0.000 }
gfCNCPoint2[7649] = {X 373.6688, Y 14.7222, Z -3.0000, A 0.000, B 0.000, C 0.000 }
gfCNCPoint2[7650] = {X 374.2467, Y 16.8917, Z -3.0000, A 0.000, B 0.000, C 0.000 }
gfCNCPoint2[7651] = {X 374.7337, Y 19.4559, Z -3.0000, A 0.000, B 0.000, C 0.000 }
gfCNCPoint2[7652] = {X 375.0386, Y 22.0481, Z -3.0000, A 0.000, B 0.000, C 0.000 }
gfCNCPoint2[7653] = {X 375.1600, Y 24.6553, Z -3.0000, A 0.000, B 0.000, C 0.000 }
gfCNCPoint2[7654] = {X 375.0972, Y 27.2646, Z -3.0000, A 0.000, B 0.000, C 0.000 }
gfCNCPoint2[7655] = {X 374.8505, Y 29.8630, Z -3.0000, A 0.000, B 0.000, C 0.000 }
gfCNCPoint2[7656] = {X 374.4212, Y 32.4374, Z -3.0000, A 0.000, B 0.000, C 0.000 }
gfCNCPoint2[7657] = {X 373.7833, Y 34.9993, Z -3.0000, A 0.000, B 0.000, C 0.000 }
gfCNCPoint2[7658] = {X 372.9218, Y 37.4948, Z -3.0000, A 0.000, B 0.000, C 0.000 }
gfCNCPoint2[7659] = {X 371.8434, Y 39.9045, Z -3.0000, A 0.000, B 0.000, C 0.000 }
gfCNCPoint2[7660] = {X 370.5564, Y 42.2096, Z -3.0000, A 0.000, B 0.000, C 0.000 }
gfCNCPoint2[7661] = {X 369.0710, Y 44.3921, Z -3.0000, A 0.000, B 0.000, C 0.000 }
gfCNCPoint2[7662] = {X 369.0323, Y 44.4442, Z -3.0000, A 0.000, B 0.000, C 0.000 }
gfCNCPoint2[7663] = {X 368.9934, Y 44.4962, Z -3.0000, A 0.000, B 0.000, C 0.000 }
gfCNCPoint2[7664] = {X 367.4735, Y 46.3510, Z -3.0000, A 0.000, B 0.000, C 0.000 }
gfCNCPoint2[7665] = {X 365.7979, Y 48.0666, Z -3.0000, A 0.000, B 0.000, C 0.000 }
gfCNCPoint2[7666] = {X 363.9795, Y 49.6299, Z -3.0000, A 0.000, B 0.000, C 0.000 }
gfCNCPoint2[7667] = {X 362.0320, Y 51.0291, Z -3.0000, A 0.000, B 0.000, C 0.000 }
gfCNCPoint2[7668] = {X 359.9702, Y 52.2536, Z -3.0000, A 0.000, B 0.000, C 0.000 }
gfCNCPoint2[7669] = {X 359.3969, Y 52.5411, Z -3.0000, A 0.000, B 0.000, C 0.000 }
gfCNCPoint2[7670] = {X 358.8172, Y 52.8153, Z -3.0000, A 0.000, B 0.000, C 0.000 }
gfCNCPoint2[7671] = {X 356.4597, Y 53.7705, Z -3.0000, A 0.000, B 0.000, C 0.000 }
gfCNCPoint2[7672] = {X 354.0251, Y 54.5078, Z -3.0000, A 0.000, B 0.000, C 0.000 }
gfCNCPoint2[7673] = {X 351.5337, Y 55.0210, Z -3.0000, A 0.000, B 0.000, C 0.000 }
gfCNCPoint2[7674] = {X 349.0060, Y 55.3059, Z -3.0000, A 0.000, B 0.000, C 0.000 }
gfCNCPoint2[7675] = {X 349.9669, Y 69.6738, Z -3.0000, A 0.000, B 0.000, C 0.000 }
gfCNCPoint2[7676] = {X 348.6528, Y 69.7412, Z -3.0000, A 0.000, B 0.000, C 0.000 }
gfCNCPoint2[7677] = {X 347.3372, Y 69.7678, Z -3.0000, A 0.000, B 0.000, C 0.000 }
gfCNCPoint2[7678] = {X 346.5719, Y 69.7765, Z -3.0000, A 0.000, B 0.000, C 0.000 }
gfCNCPoint2[7679] = {X 345.8065, Y 69.7717, Z -3.0000, A 0.000, B 0.000, C 0.000 }
gfCNCPoint2[7680] = {X 345.5896, Y 70.1915, Z -3.0000, A 0.000, B 0.000, C 0.000 }
gfCNCPoint2[7681] = {X 345.3645, Y 70.6070, Z -3.0000, A 0.000, B 0.000, C 0.000 }
gfCNCPoint2[7682] = {X 346.5773, Y 70.6173, Z -3.0000, A 0.000, B 0.000, C 0.000 }
gfCNCPoint2[7683] = {X 347.7901, Y 70.6133, Z -3.0000, A 0.000, B 0.000, C 0.000 }
gfCNCPoint2[7684] = {X 349.1241, Y 70.6191, Z -3.0000, A 0.000, B 0.000, C 0.000 }
gfCNCPoint2[7685] = {X 350.4580, Y 70.6075, Z -3.0000, A 0.000, B 0.000, C 0.000 }
gfCNCPoint2[7686] = {X 350.2073, Y 70.1433, Z -3.0000, A 0.000, B 0.000, C 0.000 }
gfCNCPoint2[7687] = {X 349.9669, Y 69.6738, Z -3.0000, A 0.000, B 0.000, C 0.000 }
gfCNCPoint2[7688] = {X 349.8068, Y 67.2792, Z -3.0000, A 0.000, B 0.000, C 0.000 }
gfCNCPoint2[7689] = {X 348.5578, Y 67.3431, Z -3.0000, A 0.000, B 0.000, C 0.000 }
gfCNCPoint2[7690] = {X 347.3074, Y 67.3679, Z -3.0000, A 0.000, B 0.000, C 0.000 }
gfCNCPoint2[7691] = {X 345.8015, Y 67.3714, Z -3.0000, A 0.000, B 0.000, C 0.000 }
gfCNCPoint2[7692] = {X 344.2965, Y 67.3197, Z -3.0000, A 0.000, B 0.000, C 0.000 }
gfCNCPoint2[7693] = {X 343.8099, Y 68.3954, Z -3.0000, A 0.000, B 0.000, C 0.000 }
gfCNCPoint2[7694] = {X 343.2656, Y 69.4431, Z -3.0000, A 0.000, B 0.000, C 0.000 }
gfCNCPoint2[7695] = {X 342.7864, Y 70.2643, Z -3.0000, A 0.000, B 0.000, C 0.000 }
gfCNCPoint2[7696] = {X 342.2717, Y 71.0638, Z -3.0000, A 0.000, B 0.000, C 0.000 }
gfCNCPoint2[7697] = {X 342.2718, Y 72.9179, Z -3.0000, A 0.000, B 0.000, C 0.000 }
gfCNCPoint2[7698] = {X 343.8005, Y 72.9735, Z -3.0000, A 0.000, B 0.000, C 0.000 }
gfCNCPoint2[7699] = {X 345.3298, Y 73.0068, Z -3.0000, A 0.000, B 0.000, C 0.000 }
gfCNCPoint2[7700] = {X 346.5590, Y 73.0173, Z -3.0000, A 0.000, B 0.000, C 0.000 }
gfCNCPoint2[7701] = {X 347.7882, Y 73.0134, Z -3.0000, A 0.000, B 0.000, C 0.000 }
gfCNCPoint2[7702] = {X 349.1414, Y 73.0190, Z -3.0000, A 0.000, B 0.000, C 0.000 }
gfCNCPoint2[7703] = {X 350.4945, Y 73.0072, Z -3.0000, A 0.000, B 0.000, C 0.000 }
gfCNCPoint2[7704] = {X 352.0276, Y 72.9726, Z -3.0000, A 0.000, B 0.000, C 0.000 }
gfCNCPoint2[7705] = {X 353.5599, Y 72.9155, Z -3.0000, A 0.000, B 0.000, C 0.000 }
gfCNCPoint2[7706] = {X 353.5598, Y 71.0781, Z -3.0000, A 0.000, B 0.000, C 0.000 }
gfCNCPoint2[7707] = {X 353.0404, Y 70.2721, Z -3.0000, A 0.000, B 0.000, C 0.000 }
gfCNCPoint2[7708] = {X 352.5571, Y 69.4440, Z -3.0000, A 0.000, B 0.000, C 0.000 }
gfCNCPoint2[7709] = {X 351.9696, Y 68.3059, Z -3.0000, A 0.000, B 0.000, C 0.000 }
gfCNCPoint2[7710] = {X 351.4503, Y 67.1351, Z -3.0000, A 0.000, B 0.000, C 0.000 }
gfCNCPoint2[7711] = {X 350.6293, Y 67.2156, Z -3.0000, A 0.000, B 0.000, C 0.000 }
gfCNCPoint2[7712] = {X 349.8068, Y 67.2792, Z -3.0000, A 0.000, B 0.000, C 0.000 }
gfCNCPoint2[7713] = {X 349.6466, Y 64.8845, Z -3.0000, A 0.000, B 0.000, C 0.000 }
gfCNCPoint2[7714] = {X 348.4628, Y 64.9450, Z -3.0000, A 0.000, B 0.000, C 0.000 }
gfCNCPoint2[7715] = {X 347.2776, Y 64.9680, Z -3.0000, A 0.000, B 0.000, C 0.000 }
gfCNCPoint2[7716] = {X 344.9731, Y 64.9481, Z -3.0000, A 0.000, B 0.000, C 0.000 }
gfCNCPoint2[7717] = {X 342.6737, Y 64.7912, Z -3.0000, A 0.000, B 0.000, C 0.000 }
gfCNCPoint2[7718] = {X 341.9389, Y 66.7262, Z -3.0000, A 0.000, B 0.000, C 0.000 }
gfCNCPoint2[7719] = {X 341.0013, Y 68.5715, Z -3.0000, A 0.000, B 0.000, C 0.000 }
gfCNCPoint2[7720] = {X 339.8716, Y 70.3059, Z -3.0000, A 0.000, B 0.000, C 0.000 }
gfCNCPoint2[7721] = {X 339.8720, Y 75.1907, Z -3.0000, A 0.000, B 0.000, C 0.000 }
gfCNCPoint2[7722] = {X 343.8270, Y 75.3752, Z -3.0000, A 0.000, B 0.000, C 0.000 }
gfCNCPoint2[7723] = {X 347.7862, Y 75.4135, Z -3.0000, A 0.000, B 0.000, C 0.000 }
gfCNCPoint2[7724] = {X 351.8753, Y 75.3780, Z -3.0000, A 0.000, B 0.000, C 0.000 }
gfCNCPoint2[7725] = {X 355.9601, Y 75.1861, Z -3.0000, A 0.000, B 0.000, C 0.000 }
gfCNCPoint2[7726] = {X 355.9597, Y 70.3191, Z -3.0000, A 0.000, B 0.000, C 0.000 }
gfCNCPoint2[7727] = {X 355.0521, Y 68.9616, Z -3.0000, A 0.000, B 0.000, C 0.000 }
gfCNCPoint2[7728] = {X 354.2626, Y 67.5321, Z -3.0000, A 0.000, B 0.000, C 0.000 }
gfCNCPoint2[7729] = {X 353.5970, Y 66.0410, Z -3.0000, A 0.000, B 0.000, C 0.000 }
gfCNCPoint2[7730] = {X 353.0598, Y 64.4989, Z -3.0000, A 0.000, B 0.000, C 0.000 }
gfCNCPoint2[7731] = {X 351.3576, Y 64.7307, Z -3.0000, A 0.000, B 0.000, C 0.000 }
gfCNCPoint2[7732] = {X 349.6466, Y 64.8845, Z -3.0000, A 0.000, B 0.000, C 0.000 }
gfCNCPoint2[7733] = {X 349.4864, Y 62.4899, Z -3.0000, A 0.000, B 0.000, C 0.000 }
gfCNCPoint2[7734] = {X 348.3678, Y 62.5468, Z -3.0000, A 0.000, B 0.000, C 0.000 }
gfCNCPoint2[7735] = {X 347.2479, Y 62.5681, Z -3.0000, A 0.000, B 0.000, C 0.000 }
gfCNCPoint2[7736] = {X 345.1177, Y 62.5519, Z -3.0000, A 0.000, B 0.000, C 0.000 }
gfCNCPoint2[7737] = {X 342.9921, Y 62.4109, Z -3.0000, A 0.000, B 0.000, C 0.000 }
gfCNCPoint2[7738] = {X 340.8784, Y 62.1457, Z -3.0000, A 0.000, B 0.000, C 0.000 }
gfCNCPoint2[7739] = {X 340.4885, Y 63.7336, Z -3.0000, A 0.000, B 0.000, C 0.000 }
gfCNCPoint2[7740] = {X 339.9471, Y 65.2766, Z -3.0000, A 0.000, B 0.000, C 0.000 }
gfCNCPoint2[7741] = {X 339.2593, Y 66.7600, Z -3.0000, A 0.000, B 0.000, C 0.000 }
gfCNCPoint2[7742] = {X 338.4316, Y 68.1701, Z -3.0000, A 0.000, B 0.000, C 0.000 }
gfCNCPoint2[7743] = {X 337.4715, Y 69.4938, Z -3.0000, A 0.000, B 0.000, C 0.000 }
gfCNCPoint2[7744] = {X 337.4721, Y 77.4162, Z -3.0000, A 0.000, B 0.000, C 0.000 }
gfCNCPoint2[7745] = {X 340.9048, Y 77.6567, Z -3.0000, A 0.000, B 0.000, C 0.000 }
gfCNCPoint2[7746] = {X 344.3433, Y 77.7892, Z -3.0000, A 0.000, B 0.000, C 0.000 }
gfCNCPoint2[7747] = {X 347.7843, Y 77.8136, Z -3.0000, A 0.000, B 0.000, C 0.000 }
gfCNCPoint2[7748] = {X 351.3134, Y 77.7927, Z -3.0000, A 0.000, B 0.000, C 0.000 }
gfCNCPoint2[7749] = {X 354.8399, Y 77.6580, Z -3.0000, A 0.000, B 0.000, C 0.000 }
gfCNCPoint2[7750] = {X 358.3603, Y 77.4095, Z -3.0000, A 0.000, B 0.000, C 0.000 }
gfCNCPoint2[7751] = {X 358.3596, Y 69.5056, Z -3.0000, A 0.000, B 0.000, C 0.000 }
gfCNCPoint2[7752] = {X 357.3486, Y 68.1061, Z -3.0000, A 0.000, B 0.000, C 0.000 }
gfCNCPoint2[7753] = {X 356.4858, Y 66.6105, Z -3.0000, A 0.000, B 0.000, C 0.000 }
gfCNCPoint2[7754] = {X 355.7802, Y 65.0347, Z -3.0000, A 0.000, B 0.000, C 0.000 }
gfCNCPoint2[7755] = {X 355.2394, Y 63.3950, Z -3.0000, A 0.000, B 0.000, C 0.000 }
gfCNCPoint2[7756] = {X 354.8689, Y 61.7086, Z -3.0000, A 0.000, B 0.000, C 0.000 }
gfCNCPoint2[7757] = {X 352.1928, Y 62.2034, Z -3.0000, A 0.000, B 0.000, C 0.000 }
gfCNCPoint2[7758] = {X 349.4864, Y 62.4899, Z -3.0000, A 0.000, B 0.000, C 0.000 }
gfCNCPoint2[7759] = {X 349.3263, Y 60.0952, Z -3.0000, A 0.000, B 0.000, C 0.000 }
gfCNCPoint2[7760] = {X 348.2728, Y 60.1487, Z -3.0000, A 0.000, B 0.000, C 0.000 }
gfCNCPoint2[7761] = {X 347.2182, Y 60.1682, Z -3.0000, A 0.000, B 0.000, C 0.000 }
gfCNCPoint2[7762] = {X 344.3864, Y 60.1133, Z -3.0000, A 0.000, B 0.000, C 0.000 }
gfCNCPoint2[7763] = {X 341.5690, Y 59.8226, Z -3.0000, A 0.000, B 0.000, C 0.000 }
gfCNCPoint2[7764] = {X 338.7856, Y 59.2982, Z -3.0000, A 0.000, B 0.000, C 0.000 }
gfCNCPoint2[7765] = {X 338.6399, Y 60.9976, Z -3.0000, A 0.000, B 0.000, C 0.000 }
gfCNCPoint2[7766] = {X 338.2959, Y 62.6682, Z -3.0000, A 0.000, B 0.000, C 0.000 }
gfCNCPoint2[7767] = {X 337.7584, Y 64.2869, Z -3.0000, A 0.000, B 0.000, C 0.000 }
gfCNCPoint2[7768] = {X 337.0347, Y 65.8314, Z -3.0000, A 0.000, B 0.000, C 0.000 }
gfCNCPoint2[7769] = {X 336.1350, Y 67.2804, Z -3.0000, A 0.000, B 0.000, C 0.000 }
gfCNCPoint2[7770] = {X 335.0715, Y 68.6139, Z -3.0000, A 0.000, B 0.000, C 0.000 }
gfCNCPoint2[7771] = {X 335.0723, Y 79.5887, Z -3.0000, A 0.000, B 0.000, C 0.000 }
gfCNCPoint2[7772] = {X 335.6732, Y 79.6587, Z -3.0000, A 0.000, B 0.000, C 0.000 }
gfCNCPoint2[7773] = {X 336.2753, Y 79.7178, Z -3.0000, A 0.000, B 0.000, C 0.000 }
gfCNCPoint2[7774] = {X 340.1046, Y 80.0147, Z -3.0000, A 0.000, B 0.000, C 0.000 }
gfCNCPoint2[7775] = {X 343.9418, Y 80.1801, Z -3.0000, A 0.000, B 0.000, C 0.000 }
gfCNCPoint2[7776] = {X 347.7824, Y 80.2137, Z -3.0000, A 0.000, B 0.000, C 0.000 }
gfCNCPoint2[7777] = {X 351.8377, Y 80.1807, Z -3.0000, A 0.000, B 0.000, C 0.000 }
gfCNCPoint2[7778] = {X 355.8892, Y 80.0006, Z -3.0000, A 0.000, B 0.000, C 0.000 }
gfCNCPoint2[7779] = {X 359.9315, Y 79.6736, Z -3.0000, A 0.000, B 0.000, C 0.000 }
gfCNCPoint2[7780] = {X 360.3463, Y 79.6320, Z -3.0000, A 0.000, B 0.000, C 0.000 }
gfCNCPoint2[7781] = {X 360.7604, Y 79.5843, Z -3.0000, A 0.000, B 0.000, C 0.000 }
gfCNCPoint2[7782] = {X 360.7596, Y 68.6242, Z -3.0000, A 0.000, B 0.000, C 0.000 }
gfCNCPoint2[7783] = {X 359.7304, Y 67.3420, Z -3.0000, A 0.000, B 0.000, C 0.000 }
gfCNCPoint2[7784] = {X 358.8533, Y 65.9514, Z -3.0000, A 0.000, B 0.000, C 0.000 }
gfCNCPoint2[7785] = {X 358.1395, Y 64.4704, Z -3.0000, A 0.000, B 0.000, C 0.000 }
gfCNCPoint2[7786] = {X 357.5981, Y 62.9179, Z -3.0000, A 0.000, B 0.000, C 0.000 }
gfCNCPoint2[7787] = {X 357.2362, Y 61.3142, Z -3.0000, A 0.000, B 0.000, C 0.000 }
gfCNCPoint2[7788] = {X 357.0917, Y 60.1647, Z -3.0000, A 0.000, B 0.000, C 0.000 }
gfCNCPoint2[7789] = {X 357.0395, Y 59.0073, Z -3.0000, A 0.000, B 0.000, C 0.000 }
gfCNCPoint2[7790] = {X 357.0394, Y 58.6377, Z -3.0000, A 0.000, B 0.000, C 0.000 }
gfCNCPoint2[7791] = {X 355.6983, Y 59.0312, Z -3.0000, A 0.000, B 0.000, C 0.000 }
gfCNCPoint2[7792] = {X 354.3416, Y 59.3673, Z -3.0000, A 0.000, B 0.000, C 0.000 }
gfCNCPoint2[7793] = {X 351.8480, Y 59.8283, Z -3.0000, A 0.000, B 0.000, C 0.000 }
gfCNCPoint2[7794] = {X 349.3263, Y 60.0952, Z -3.0000, A 0.000, B 0.000, C 0.000 }
gfCNCPoint2[7795] = {X 349.1661, Y 57.7006, Z -3.0000, A 0.000, B 0.000, C 0.000 }
gfCNCPoint2[7796] = {X 348.1779, Y 57.7505, Z -3.0000, A 0.000, B 0.000, C 0.000 }
gfCNCPoint2[7797] = {X 347.1885, Y 57.7683, Z -3.0000, A 0.000, B 0.000, C 0.000 }
gfCNCPoint2[7798] = {X 344.5488, Y 57.7187, Z -3.0000, A 0.000, B 0.000, C 0.000 }
gfCNCPoint2[7799] = {X 341.9225, Y 57.4487, Z -3.0000, A 0.000, B 0.000, C 0.000 }
gfCNCPoint2[7800] = {X 339.3279, Y 56.9602, Z -3.0000, A 0.000, B 0.000, C 0.000 }
gfCNCPoint2[7801] = {X 337.7708, Y 56.5570, Z -3.0000, A 0.000, B 0.000, C 0.000 }
gfCNCPoint2[7802] = {X 336.2363, Y 56.0750, Z -3.0000, A 0.000, B 0.000, C 0.000 }
gfCNCPoint2[7803] = {X 336.3520, Y 57.0344, Z -3.0000, A 0.000, B 0.000, C 0.000 }
gfCNCPoint2[7804] = {X 336.3907, Y 58.0000, Z -3.0000, A 0.000, B 0.000, C 0.000 }
gfCNCPoint2[7805] = {X 336.3907, Y 58.9493, Z -3.0000, A 0.000, B 0.000, C 0.000 }
gfCNCPoint2[7806] = {X 336.3894, Y 59.0917, Z -3.0000, A 0.000, B 0.000, C 0.000 }
gfCNCPoint2[7807] = {X 336.3864, Y 59.2340, Z -3.0000, A 0.000, B 0.000, C 0.000 }
gfCNCPoint2[7808] = {X 336.2427, Y 60.7983, Z -3.0000, A 0.000, B 0.000, C 0.000 }
gfCNCPoint2[7809] = {X 335.8979, Y 62.3308, Z -3.0000, A 0.000, B 0.000, C 0.000 }
gfCNCPoint2[7810] = {X 335.3577, Y 63.8059, Z -3.0000, A 0.000, B 0.000, C 0.000 }
gfCNCPoint2[7811] = {X 334.6313, Y 65.1988, Z -3.0000, A 0.000, B 0.000, C 0.000 }
gfCNCPoint2[7812] = {X 333.7308, Y 66.4859, Z -3.0000, A 0.000, B 0.000, C 0.000 }
gfCNCPoint2[7813] = {X 332.6714, Y 67.6458, Z -3.0000, A 0.000, B 0.000, C 0.000 }
gfCNCPoint2[7814] = {X 332.6725, Y 81.6423, Z -3.0000, A 0.000, B 0.000, C 0.000 }
gfCNCPoint2[7815] = {X 334.3584, Y 81.9154, Z -3.0000, A 0.000, B 0.000, C 0.000 }
gfCNCPoint2[7816] = {X 336.0555, Y 82.1077, Z -3.0000, A 0.000, B 0.000, C 0.000 }
gfCNCPoint2[7817] = {X 339.9573, Y 82.4102, Z -3.0000, A 0.000, B 0.000, C 0.000 }
gfCNCPoint2[7818] = {X 343.8671, Y 82.5790, Z -3.0000, A 0.000, B 0.000, C 0.000 }
gfCNCPoint2[7819] = {X 347.7804, Y 82.6138, Z -3.0000, A 0.000, B 0.000, C 0.000 }
gfCNCPoint2[7820] = {X 351.9132, Y 82.5796, Z -3.0000, A 0.000, B 0.000, C 0.000 }
gfCNCPoint2[7821] = {X 356.0420, Y 82.3958, Z -3.0000, A 0.000, B 0.000, C 0.000 }
gfCNCPoint2[7822] = {X 360.1614, Y 82.0626, Z -3.0000, A 0.000, B 0.000, C 0.000 }
gfCNCPoint2[7823] = {X 361.6662, Y 81.8850, Z -3.0000, A 0.000, B 0.000, C 0.000 }
gfCNCPoint2[7824] = {X 363.1606, Y 81.6342, Z -3.0000, A 0.000, B 0.000, C 0.000 }
gfCNCPoint2[7825] = {X 363.1595, Y 67.6542, Z -3.0000, A 0.000, B 0.000, C 0.000 }
gfCNCPoint2[7826] = {X 362.0732, Y 66.4639, Z -3.0000, A 0.000, B 0.000, C 0.000 }
gfCNCPoint2[7827] = {X 361.1550, Y 65.1396, Z -3.0000, A 0.000, B 0.000, C 0.000 }
gfCNCPoint2[7828] = {X 360.4213, Y 63.7049, Z -3.0000, A 0.000, B 0.000, C 0.000 }
gfCNCPoint2[7829] = {X 359.8850, Y 62.1852, Z -3.0000, A 0.000, B 0.000, C 0.000 }
gfCNCPoint2[7830] = {X 359.5558, Y 60.6078, Z -3.0000, A 0.000, B 0.000, C 0.000 }
gfCNCPoint2[7831] = {X 359.4395, Y 59.0005, Z -3.0000, A 0.000, B 0.000, C 0.000 }
gfCNCPoint2[7832] = {X 359.4393, Y 58.0000, Z -3.0000, A 0.000, B 0.000, C 0.000 }
gfCNCPoint2[7833] = {X 359.5345, Y 56.4863, Z -3.0000, A 0.000, B 0.000, C 0.000 }
gfCNCPoint2[7834] = {X 359.8187, Y 54.9964, Z -3.0000, A 0.000, B 0.000, C 0.000 }
gfCNCPoint2[7835] = {X 358.0876, Y 55.7273, Z -3.0000, A 0.000, B 0.000, C 0.000 }
gfCNCPoint2[7836] = {X 356.3147, Y 56.3497, Z -3.0000, A 0.000, B 0.000, C 0.000 }
gfCNCPoint2[7837] = {X 353.9704, Y 56.9903, Z -3.0000, A 0.000, B 0.000, C 0.000 }
gfCNCPoint2[7838] = {X 351.5825, Y 57.4416, Z -3.0000, A 0.000, B 0.000, C 0.000 }
gfCNCPoint2[7839] = {X 349.1661, Y 57.7006, Z -3.0000, A 0.000, B 0.000, C 0.000 }
gfCNCPoint2[7840] = {X 349.0060, Y 55.3059, Z -3.0000, A 0.000, B 0.000, C 0.000 }
gfCNCPoint2[7841] = {X 348.0829, Y 55.3524, Z -3.0000, A 0.000, B 0.000, C 0.000 }
gfCNCPoint2[7842] = {X 347.1589, Y 55.3683, Z -3.0000, A 0.000, B 0.000, C 0.000 }
gfCNCPoint2[7843] = {X 344.5805, Y 55.3160, Z -3.0000, A 0.000, B 0.000, C 0.000 }
gfCNCPoint2[7844] = {X 342.0169, Y 55.0362, Z -3.0000, A 0.000, B 0.000, C 0.000 }
gfCNCPoint2[7845] = {X 339.4880, Y 54.5310, Z -3.0000, A 0.000, B 0.000, C 0.000 }
gfCNCPoint2[7846] = {X 337.0137, Y 53.8044, Z -3.0000, A 0.000, B 0.000, C 0.000 }
gfCNCPoint2[7847] = {X 334.7573, Y 52.9257, Z -3.0000, A 0.000, B 0.000, C 0.000 }
gfCNCPoint2[7848] = {X 332.5817, Y 51.8629, Z -3.0000, A 0.000, B 0.000, C 0.000 }
gfCNCPoint2[7849] = {X 331.5843, Y 51.2764, Z -3.0000, A 0.000, B 0.000, C 0.000 }
gfCNCPoint2[7850] = {X 330.6109, Y 50.6508, Z -3.0000, A 0.000, B 0.000, C 0.000 }
gfCNCPoint2[7851] = {X 331.5774, Y 51.6049, Z -3.0000, A 0.000, B 0.000, C 0.000 }
gfCNCPoint2[7852] = {X 332.4009, Y 52.6848, Z -3.0000, A 0.000, B 0.000, C 0.000 }
gfCNCPoint2[7853] = {X 333.0651, Y 53.8694, Z -3.0000, A 0.000, B 0.000, C 0.000 }
gfCNCPoint2[7854] = {X 333.5571, Y 55.1352, Z -3.0000, A 0.000, B 0.000, C 0.000 }
gfCNCPoint2[7855] = {X 333.8670, Y 56.4574, Z -3.0000, A 0.000, B 0.000, C 0.000 }
gfCNCPoint2[7856] = {X 333.9597, Y 57.2262, Z -3.0000, A 0.000, B 0.000, C 0.000 }
gfCNCPoint2[7857] = {X 333.9907, Y 58.0000, Z -3.0000, A 0.000, B 0.000, C 0.000 }
gfCNCPoint2[7858] = {X 333.9907, Y 58.9450, Z -3.0000, A 0.000, B 0.000, C 0.000 }
gfCNCPoint2[7859] = {X 333.8758, Y 60.4000, Z -3.0000, A 0.000, B 0.000, C 0.000 }
gfCNCPoint2[7860] = {X 333.5444, Y 61.8214, Z -3.0000, A 0.000, B 0.000, C 0.000 }
gfCNCPoint2[7861] = {X 333.0039, Y 63.1771, Z -3.0000, A 0.000, B 0.000, C 0.000 }
gfCNCPoint2[7862] = {X 332.2664, Y 64.4366, Z -3.0000, A 0.000, B 0.000, C 0.000 }
gfCNCPoint2[7863] = {X 331.3487, Y 65.5715, Z -3.0000, A 0.000, B 0.000, C 0.000 }
gfCNCPoint2[7864] = {X 330.2713, Y 66.5561, Z -3.0000, A 0.000, B 0.000, C 0.000 }
gfCNCPoint2[7865] = {X 330.2726, Y 83.2031, Z -3.0000, A 0.000, B 0.000, C 0.000 }
gfCNCPoint2[7866] = {X 330.2763, Y 83.5834, Z -3.0000, A 0.000, B 0.000, C 0.000 }
gfCNCPoint2[7867] = {X 330.3821, Y 83.6086, Z -3.0000, A 0.000, B 0.000, C 0.000 }
gfCNCPoint2[7868] = {X 333.0927, Y 84.1520, Z -3.0000, A 0.000, B 0.000, C 0.000 }
gfCNCPoint2[7869] = {X 335.8356, Y 84.4976, Z -3.0000, A 0.000, B 0.000, C 0.000 }
gfCNCPoint2[7870] = {X 339.8099, Y 84.8057, Z -3.0000, A 0.000, B 0.000, C 0.000 }
gfCNCPoint2[7871] = {X 343.7924, Y 84.9778, Z -3.0000, A 0.000, B 0.000, C 0.000 }
gfCNCPoint2[7872] = {X 347.7785, Y 85.0139, Z -3.0000, A 0.000, B 0.000, C 0.000 }
gfCNCPoint2[7873] = {X 351.9887, Y 84.9784, Z -3.0000, A 0.000, B 0.000, C 0.000 }
gfCNCPoint2[7874] = {X 356.1948, Y 84.7909, Z -3.0000, A 0.000, B 0.000, C 0.000 }
gfCNCPoint2[7875] = {X 360.3914, Y 84.4516, Z -3.0000, A 0.000, B 0.000, C 0.000 }
gfCNCPoint2[7876] = {X 362.9937, Y 84.1047, Z -3.0000, A 0.000, B 0.000, C 0.000 }
gfCNCPoint2[7877] = {X 365.5607, Y 83.5546, Z -3.0000, A 0.000, B 0.000, C 0.000 }
gfCNCPoint2[7878] = {X 365.5594, Y 66.5618, Z -3.0000, A 0.000, B 0.000, C 0.000 }
gfCNCPoint2[7879] = {X 364.4848, Y 65.5838, Z -3.0000, A 0.000, B 0.000, C 0.000 }
gfCNCPoint2[7880] = {X 363.5688, Y 64.4560, Z -3.0000, A 0.000, B 0.000, C 0.000 }
gfCNCPoint2[7881] = {X 362.8318, Y 63.2038, Z -3.0000, A 0.000, B 0.000, C 0.000 }
gfCNCPoint2[7882] = {X 362.2906, Y 61.8554, Z -3.0000, A 0.000, B 0.000, C 0.000 }
gfCNCPoint2[7883] = {X 361.9573, Y 60.4412, Z -3.0000, A 0.000, B 0.000, C 0.000 }
gfCNCPoint2[7884] = {X 361.8395, Y 58.9930, Z -3.0000, A 0.000, B 0.000, C 0.000 }
gfCNCPoint2[7885] = {X 361.8393, Y 58.0000, Z -3.0000, A 0.000, B 0.000, C 0.000 }
gfCNCPoint2[7886] = {X 361.9156, Y 56.7870, Z -3.0000, A 0.000, B 0.000, C 0.000 }
gfCNCPoint2[7887] = {X 362.1433, Y 55.5931, Z -3.0000, A 0.000, B 0.000, C 0.000 }
gfCNCPoint2[7888] = {X 362.5747, Y 54.2990, Z -3.0000, A 0.000, B 0.000, C 0.000 }
gfCNCPoint2[7889] = {X 363.1838, Y 53.0783, Z -3.0000, A 0.000, B 0.000, C 0.000 }
gfCNCPoint2[7890] = {X 363.9585, Y 51.9554, Z -3.0000, A 0.000, B 0.000, C 0.000 }
gfCNCPoint2[7891] = {X 364.8833, Y 50.9526, Z -3.0000, A 0.000, B 0.000, C 0.000 }
gfCNCPoint2[7892] = {X 365.9399, Y 50.0897, Z -3.0000, A 0.000, B 0.000, C 0.000 }
gfCNCPoint2[7893] = {X 367.1073, Y 49.3839, Z -3.0000, A 0.000, B 0.000, C 0.000 }
gfCNCPoint2[7894] = {X 368.3624, Y 48.8492, Z -3.0000, A 0.000, B 0.000, C 0.000 }
gfCNCPoint2[7895] = {X 369.6801, Y 48.4963, Z -3.0000, A 0.000, B 0.000, C 0.000 }
gfCNCPoint2[7896] = {X 371.0344, Y 48.3322, Z -3.0000, A 0.000, B 0.000, C 0.000 }
gfCNCPoint2[7897] = {X 371.2768, Y 48.3230, Z -3.0000, A 0.000, B 0.000, C 0.000 }
gfCNCPoint2[7898] = {X 371.5193, Y 48.3200, Z -3.0000, A 0.000, B 0.000, C 0.000 }
gfCNCPoint2[7899] = {X 388.0597, Y 48.3200, Z -3.0000, A 0.000, B 0.000, C 0.000 }
gfCNCPoint2[7900] = {X 389.4419, Y 48.4192, Z -3.0000, A 0.000, B 0.000, C 0.000 }
gfCNCPoint2[7901] = {X 390.7958, Y 48.7147, Z -3.0000, A 0.000, B 0.000, C 0.000 }
gfCNCPoint2[7902] = {X 392.0936, Y 49.2006, Z -3.0000, A 0.000, B 0.000, C 0.000 }
gfCNCPoint2[7903] = {X 393.3087, Y 49.8667, Z -3.0000, A 0.000, B 0.000, C 0.000 }
gfCNCPoint2[7904] = {X 394.5333, Y 49.1962, Z -3.0000, A 0.000, B 0.000, C 0.000 }
gfCNCPoint2[7905] = {X 395.8416, Y 48.7089, Z -3.0000, A 0.000, B 0.000, C 0.000 }
gfCNCPoint2[7906] = {X 397.1858, Y 48.4177, Z -3.0000, A 0.000, B 0.000, C 0.000 }
gfCNCPoint2[7907] = {X 398.5577, Y 48.3200, Z -3.0000, A 0.000, B 0.000, C 0.000 }
gfCNCPoint2[7908] = {X 398.7346, Y 48.3200, Z -3.0000, A 0.000, B 0.000, C 0.000 }
gfCNCPoint2[7909] = {X 398.1859, Y 47.6069, Z -3.0000, A 0.000, B 0.000, C 0.000 }
gfCNCPoint2[7910] = {X 397.7774, Y 46.8051, Z -3.0000, A 0.000, B 0.000, C 0.000 }
gfCNCPoint2[7911] = {X 397.5230, Y 45.9420, Z -3.0000, A 0.000, B 0.000, C 0.000 }
gfCNCPoint2[7912] = {X 397.4561, Y 45.4921, Z -3.0000, A 0.000, B 0.000, C 0.000 }
gfCNCPoint2[7913] = {X 397.4314, Y 45.0378, Z -3.0000, A 0.000, B 0.000, C 0.000 }
gfCNCPoint2[7914] = {X 397.4316, Y 44.1456, Z -3.0000, A 0.000, B 0.000, C 0.000 }
gfCNCPoint2[7915] = {X 397.5413, Y 43.1780, Z -3.0000, A 0.000, B 0.000, C 0.000 }
gfCNCPoint2[7916] = {X 397.8410, Y 42.2514, Z -3.0000, A 0.000, B 0.000, C 0.000 }
gfCNCPoint2[7917] = {X 398.3186, Y 41.4029, Z -3.0000, A 0.000, B 0.000, C 0.000 }
gfCNCPoint2[7918] = {X 398.9552, Y 40.6660, Z -3.0000, A 0.000, B 0.000, C 0.000 }
gfCNCPoint2[7919] = {X 398.9552, Y 31.8223, Z -3.0000, A 0.000, B 0.000, C 0.000 }
gfCNCPoint2[7920] = {X 396.7484, Y 27.9866, Z -3.0000, A 0.000, B 0.000, C 0.000 }
gfCNCPoint2[7921] = {X 386.3470, Y 33.9707, Z -3.0000, A 0.000, B 0.000, C 0.000 }
gfCNCPoint2[7922] = {X 386.2661, Y 34.3977, Z -3.0000, A 0.000, B 0.000, C 0.000 }
gfCNCPoint2[7923] = {X 386.1815, Y 34.8239, Z -3.0000, A 0.000, B 0.000, C 0.000 }
gfCNCPoint2[7924] = {X 386.0225, Y 35.5735, Z -3.0000, A 0.000, B 0.000, C 0.000 }
gfCNCPoint2[7925] = {X 385.8497, Y 36.3200, Z -3.0000, A 0.000, B 0.000, C 0.000 }
gfCNCPoint2[7926] = {X 386.9552, Y 36.3200, Z -3.0000, A 0.000, B 0.000, C 0.000 }
gfCNCPoint2[7927] = {X 386.9552, Y 35.0279, Z -3.0000, A 0.000, B 0.000, C 0.000 }
gfCNCPoint2[7928] = {X 386.3470, Y 33.9707, Z -3.0000, A 0.000, B 0.000, C 0.000 }
gfCNCPoint2[7929] = {X 388.4273, Y 32.7739, Z -3.0000, A 0.000, B 0.000, C 0.000 }
gfCNCPoint2[7930] = {X 386.4752, Y 29.3809, Z -3.0000, A 0.000, B 0.000, C 0.000 }
gfCNCPoint2[7931] = {X 384.7444, Y 26.3627, Z -3.0000, A 0.000, B 0.000, C 0.000 }
gfCNCPoint2[7932] = {X 384.6156, Y 28.7653, Z -3.0000, A 0.000, B 0.000, C 0.000 }
gfCNCPoint2[7933] = {X 384.3629, Y 31.1581, Z -3.0000, A 0.000, B 0.000, C 0.000 }
gfCNCPoint2[7934] = {X 383.9869, Y 33.5347, Z -3.0000, A 0.000, B 0.000, C 0.000 }
gfCNCPoint2[7935] = {X 383.9100, Y 33.9410, Z -3.0000, A 0.000, B 0.000, C 0.000 }
gfCNCPoint2[7936] = {X 383.8294, Y 34.3466, Z -3.0000, A 0.000, B 0.000, C 0.000 }
gfCNCPoint2[7937] = {X 383.6795, Y 35.0535, Z -3.0000, A 0.000, B 0.000, C 0.000 }
gfCNCPoint2[7938] = {X 383.5166, Y 35.7576, Z -3.0000, A 0.000, B 0.000, C 0.000 }
gfCNCPoint2[7939] = {X 383.1267, Y 37.2470, Z -3.0000, A 0.000, B 0.000, C 0.000 }
gfCNCPoint2[7940] = {X 382.6790, Y 38.7200, Z -3.0000, A 0.000, B 0.000, C 0.000 }
gfCNCPoint2[7941] = {X 388.0597, Y 38.7200, Z -3.0000, A 0.000, B 0.000, C 0.000 }
gfCNCPoint2[7942] = {X 388.4821, Y 38.7246, Z -3.0000, A 0.000, B 0.000, C 0.000 }
gfCNCPoint2[7943] = {X 388.9043, Y 38.7385, Z -3.0000, A 0.000, B 0.000, C 0.000 }
gfCNCPoint2[7944] = {X 389.1204, Y 38.2363, Z -3.0000, A 0.000, B 0.000, C 0.000 }
gfCNCPoint2[7945] = {X 389.3552, Y 37.7427, Z -3.0000, A 0.000, B 0.000, C 0.000 }
gfCNCPoint2[7946] = {X 389.3552, Y 34.3867, Z -3.0000, A 0.000, B 0.000, C 0.000 }
gfCNCPoint2[7947] = {X 388.4273, Y 32.7739, Z -3.0000, A 0.000, B 0.000, C 0.000 }
gfCNCPoint2[7948] = {X 390.5076, Y 31.5771, Z -3.0000, A 0.000, B 0.000, C 0.000 }
gfCNCPoint2[7949] = {X 388.5564, Y 28.1855, Z -3.0000, A 0.000, B 0.000, C 0.000 }
gfCNCPoint2[7950] = {X 386.8253, Y 25.1670, Z -3.0000, A 0.000, B 0.000, C 0.000 }
gfCNCPoint2[7951] = {X 386.1701, Y 24.0480, Z -3.0000, A 0.000, B 0.000, C 0.000 }
gfCNCPoint2[7952] = {X 385.4967, Y 22.9398, Z -3.0000, A 0.000, B 0.000, C 0.000 }
gfCNCPoint2[7953] = {X 384.4685, Y 22.1502, Z -3.0000, A 0.000, B 0.000, C 0.000 }
gfCNCPoint2[7954] = {X 383.5309, Y 21.2550, Z -3.0000, A 0.000, B 0.000, C 0.000 }
gfCNCPoint2[7955] = {X 382.6946, Y 20.2645, Z -3.0000, A 0.000, B 0.000, C 0.000 }
gfCNCPoint2[7956] = {X 381.9693, Y 19.1900, Z -3.0000, A 0.000, B 0.000, C 0.000 }
gfCNCPoint2[7957] = {X 382.2219, Y 21.5509, Z -3.0000, A 0.000, B 0.000, C 0.000 }
gfCNCPoint2[7958] = {X 382.3474, Y 23.9218, Z -3.0000, A 0.000, B 0.000, C 0.000 }
gfCNCPoint2[7959] = {X 382.3453, Y 26.2961, Z -3.0000, A 0.000, B 0.000, C 0.000 }
gfCNCPoint2[7960] = {X 382.2016, Y 28.8358, Z -3.0000, A 0.000, B 0.000, C 0.000 }
gfCNCPoint2[7961] = {X 381.9120, Y 31.3630, Z -3.0000, A 0.000, B 0.000, C 0.000 }
gfCNCPoint2[7962] = {X 381.4774, Y 33.8694, Z -3.0000, A 0.000, B 0.000, C 0.000 }
gfCNCPoint2[7963] = {X 380.9959, Y 35.9389, Z -3.0000, A 0.000, B 0.000, C 0.000 }
gfCNCPoint2[7964] = {X 380.3967, Y 37.9775, Z -3.0000, A 0.000, B 0.000, C 0.000 }
gfCNCPoint2[7965] = {X 379.8412, Y 39.5621, Z -3.0000, A 0.000, B 0.000, C 0.000 }
gfCNCPoint2[7966] = {X 379.2145, Y 41.1200, Z -3.0000, A 0.000, B 0.000, C 0.000 }
gfCNCPoint2[7967] = {X 388.0597, Y 41.1200, Z -3.0000, A 0.000, B 0.000, C 0.000 }
gfCNCPoint2[7968] = {X 389.3256, Y 41.1675, Z -3.0000, A 0.000, B 0.000, C 0.000 }
gfCNCPoint2[7969] = {X 390.5843, Y 41.3099, Z -3.0000, A 0.000, B 0.000, C 0.000 }
gfCNCPoint2[7970] = {X 391.0709, Y 39.7838, Z -3.0000, A 0.000, B 0.000, C 0.000 }
gfCNCPoint2[7971] = {X 391.7552, Y 38.3355, Z -3.0000, A 0.000, B 0.000, C 0.000 }
gfCNCPoint2[7972] = {X 391.7552, Y 33.7456, Z -3.0000, A 0.000, B 0.000, C 0.000 }
gfCNCPoint2[7973] = {X 390.5076, Y 31.5771, Z -3.0000, A 0.000, B 0.000, C 0.000 }
gfCNCPoint2[7974] = {X 392.5879, Y 30.3802, Z -3.0000, A 0.000, B 0.000, C 0.000 }
gfCNCPoint2[7975] = {X 390.6375, Y 26.9902, Z -3.0000, A 0.000, B 0.000, C 0.000 }
gfCNCPoint2[7976] = {X 388.9417, Y 24.0330, Z -3.0000, A 0.000, B 0.000, C 0.000 }
gfCNCPoint2[7977] = {X 388.1112, Y 22.6179, Z -3.0000, A 0.000, B 0.000, C 0.000 }
gfCNCPoint2[7978] = {X 387.2524, Y 21.2197, Z -3.0000, A 0.000, B 0.000, C 0.000 }
gfCNCPoint2[7979] = {X 386.3051, Y 20.5548, Z -3.0000, A 0.000, B 0.000, C 0.000 }
gfCNCPoint2[7980] = {X 385.4439, Y 19.7816, Z -3.0000, A 0.000, B 0.000, C 0.000 }
gfCNCPoint2[7981] = {X 384.6811, Y 18.9111, Z -3.0000, A 0.000, B 0.000, C 0.000 }
gfCNCPoint2[7982] = {X 384.0276, Y 17.9559, Z -3.0000, A 0.000, B 0.000, C 0.000 }
gfCNCPoint2[7983] = {X 383.4396, Y 16.8082, Z -3.0000, A 0.000, B 0.000, C 0.000 }
gfCNCPoint2[7984] = {X 383.0094, Y 15.5925, Z -3.0000, A 0.000, B 0.000, C 0.000 }
gfCNCPoint2[7985] = {X 382.7446, Y 14.3304, Z -3.0000, A 0.000, B 0.000, C 0.000 }
gfCNCPoint2[7986] = {X 382.6498, Y 13.0443, Z -3.0000, A 0.000, B 0.000, C 0.000 }
gfCNCPoint2[7987] = {X 382.6496, Y 12.1868, Z -3.0000, A 0.000, B 0.000, C 0.000 }
gfCNCPoint2[7988] = {X 382.6507, Y 12.0459, Z -3.0000, A 0.000, B 0.000, C 0.000 }
gfCNCPoint2[7989] = {X 382.6537, Y 11.9050, Z -3.0000, A 0.000, B 0.000, C 0.000 }
gfCNCPoint2[7990] = {X 377.7923, Y 11.9050, Z -3.0000, A 0.000, B 0.000, C 0.000 }
gfCNCPoint2[7991] = {X 378.4176, Y 13.8510, Z -3.0000, A 0.000, B 0.000, C 0.000 }
gfCNCPoint2[7992] = {X 378.9278, Y 15.8302, Z -3.0000, A 0.000, B 0.000, C 0.000 }
gfCNCPoint2[7993] = {X 379.3004, Y 17.6624, Z -3.0000, A 0.000, B 0.000, C 0.000 }
gfCNCPoint2[7994] = {X 379.5906, Y 19.5095, Z -3.0000, A 0.000, B 0.000, C 0.000 }
gfCNCPoint2[7995] = {X 379.8694, Y 22.2860, Z -3.0000, A 0.000, B 0.000, C 0.000 }
gfCNCPoint2[7996] = {X 379.9623, Y 25.0750, Z -3.0000, A 0.000, B 0.000, C 0.000 }
gfCNCPoint2[7997] = {X 379.8688, Y 27.8639, Z -3.0000, A 0.000, B 0.000, C 0.000 }
gfCNCPoint2[7998] = {X 379.5894, Y 30.6404, Z -3.0000, A 0.000, B 0.000, C 0.000 }
gfCNCPoint2[7999] = {X 379.1253, Y 33.3921, Z -3.0000, A 0.000, B 0.000, C 0.000 }
gfCNCPoint2[8000] = {X 378.5751, Y 35.6993, Z -3.0000, A 0.000, B 0.000, C 0.000 }
gfCNCPoint2[8001] = {X 377.8685, Y 37.9635, Z -3.0000, A 0.000, B 0.000, C 0.000 }
gfCNCPoint2[8002] = {X 377.0088, Y 40.1741, Z -3.0000, A 0.000, B 0.000, C 0.000 }
gfCNCPoint2[8003] = {X 376.2271, Y 41.8693, Z -3.0000, A 0.000, B 0.000, C 0.000 }
gfCNCPoint2[8004] = {X 375.3554, Y 43.5200, Z -3.0000, A 0.000, B 0.000, C 0.000 }
gfCNCPoint2[8005] = {X 388.0597, Y 43.5200, Z -3.0000, A 0.000, B 0.000, C 0.000 }
gfCNCPoint2[8006] = {X 389.6072, Y 43.6029, Z -3.0000, A 0.000, B 0.000, C 0.000 }
gfCNCPoint2[8007] = {X 391.1370, Y 43.8508, Z -3.0000, A 0.000, B 0.000, C 0.000 }
gfCNCPoint2[8008] = {X 392.6316, Y 44.2607, Z -3.0000, A 0.000, B 0.000, C 0.000 }
gfCNCPoint2[8009] = {X 392.7236, Y 42.8756, Z -3.0000, A 0.000, B 0.000, C 0.000 }
gfCNCPoint2[8010] = {X 393.0129, Y 41.5179, Z -3.0000, A 0.000, B 0.000, C 0.000 }
gfCNCPoint2[8011] = {X 393.4934, Y 40.2155, Z -3.0000, A 0.000, B 0.000, C 0.000 }
gfCNCPoint2[8012] = {X 394.1552, Y 38.9952, Z -3.0000, A 0.000, B 0.000, C 0.000 }
gfCNCPoint2[8013] = {X 394.1552, Y 33.1045, Z -3.0000, A 0.000, B 0.000, C 0.000 }
gfCNCPoint2[8014] = {X 392.5879, Y 30.3802, Z -3.0000, A 0.000, B 0.000, C 0.000 }
gfCNCPoint2[8015] = {X 394.6681, Y 29.1834, Z -3.0000, A 0.000, B 0.000, C 0.000 }
gfCNCPoint2[8016] = {X 392.7186, Y 25.7948, Z -3.0000, A 0.000, B 0.000, C 0.000 }
gfCNCPoint2[8017] = {X 391.0237, Y 22.8391, Z -3.0000, A 0.000, B 0.000, C 0.000 }
gfCNCPoint2[8018] = {X 390.1123, Y 21.2885, Z -3.0000, A 0.000, B 0.000, C 0.000 }
gfCNCPoint2[8019] = {X 389.1680, Y 19.7577, Z -3.0000, A 0.000, B 0.000, C 0.000 }
gfCNCPoint2[8020] = {X 389.0448, Y 19.5768, Z -3.0000, A 0.000, B 0.000, C 0.000 }
gfCNCPoint2[8021] = {X 388.9095, Y 19.4046, Z -3.0000, A 0.000, B 0.000, C 0.000 }
gfCNCPoint2[8022] = {X 387.8200, Y 18.6930, Z -3.0000, A 0.000, B 0.000, C 0.000 }
gfCNCPoint2[8023] = {X 386.8745, Y 17.7988, Z -3.0000, A 0.000, B 0.000, C 0.000 }
gfCNCPoint2[8024] = {X 386.1034, Y 16.7506, Z -3.0000, A 0.000, B 0.000, C 0.000 }
gfCNCPoint2[8025] = {X 385.5312, Y 15.5818, Z -3.0000, A 0.000, B 0.000, C 0.000 }
gfCNCPoint2[8026] = {X 385.1762, Y 14.3298, Z -3.0000, A 0.000, B 0.000, C 0.000 }
gfCNCPoint2[8027] = {X 385.0498, Y 13.0347, Z -3.0000, A 0.000, B 0.000, C 0.000 }
gfCNCPoint2[8028] = {X 385.0496, Y 12.1868, Z -3.0000, A 0.000, B 0.000, C 0.000 }
gfCNCPoint2[8029] = {X 385.0504, Y 12.0808, Z -3.0000, A 0.000, B 0.000, C 0.000 }
gfCNCPoint2[8030] = {X 385.0527, Y 11.9749, Z -3.0000, A 0.000, B 0.000, C 0.000 }
gfCNCPoint2[8031] = {X 385.1994, Y 10.7178, Z -3.0000, A 0.000, B 0.000, C 0.000 }
gfCNCPoint2[8032] = {X 385.5616, Y 9.5050, Z -3.0000, A 0.000, B 0.000, C 0.000 }
gfCNCPoint2[8033] = {X 374.2007, Y 9.5050, Z -3.0000, A 0.000, B 0.000, C 0.000 }
gfCNCPoint2[8034] = {X 374.9080, Y 11.0877, Z -3.0000, A 0.000, B 0.000, C 0.000 }
gfCNCPoint2[8035] = {X 375.5299, Y 12.7059, Z -3.0000, A 0.000, B 0.000, C 0.000 }
gfCNCPoint2[8036] = {X 376.1121, Y 14.5179, Z -3.0000, A 0.000, B 0.000, C 0.000 }
gfCNCPoint2[8037] = {X 376.5872, Y 16.3610, Z -3.0000, A 0.000, B 0.000, C 0.000 }
gfCNCPoint2[8038] = {X 377.1058, Y 19.0915, Z -3.0000, A 0.000, B 0.000, C 0.000 }
gfCNCPoint2[8039] = {X 377.4306, Y 21.8517, Z -3.0000, A 0.000, B 0.000, C 0.000 }
gfCNCPoint2[8040] = {X 377.5598, Y 24.6280, Z -3.0000, A 0.000, B 0.000, C 0.000 }
gfCNCPoint2[8041] = {X 377.4930, Y 27.4065, Z -3.0000, A 0.000, B 0.000, C 0.000 }
gfCNCPoint2[8042] = {X 377.2304, Y 30.1734, Z -3.0000, A 0.000, B 0.000, C 0.000 }
gfCNCPoint2[8043] = {X 376.7733, Y 32.9148, Z -3.0000, A 0.000, B 0.000, C 0.000 }
gfCNCPoint2[8044] = {X 376.1757, Y 35.3676, Z -3.0000, A 0.000, B 0.000, C 0.000 }
gfCNCPoint2[8045] = {X 375.3882, Y 37.7662, Z -3.0000, A 0.000, B 0.000, C 0.000 }
gfCNCPoint2[8046] = {X 374.4157, Y 40.0959, Z -3.0000, A 0.000, B 0.000, C 0.000 }
gfCNCPoint2[8047] = {X 373.2641, Y 42.3425, Z -3.0000, A 0.000, B 0.000, C 0.000 }
gfCNCPoint2[8048] = {X 372.1862, Y 44.1205, Z -3.0000, A 0.000, B 0.000, C 0.000 }
gfCNCPoint2[8049] = {X 370.9960, Y 45.8254, Z -3.0000, A 0.000, B 0.000, C 0.000 }
gfCNCPoint2[8050] = {X 370.9142, Y 45.9352, Z -3.0000, A 0.000, B 0.000, C 0.000 }
gfCNCPoint2[8051] = {X 371.2166, Y 45.9238, Z -3.0000, A 0.000, B 0.000, C 0.000 }
gfCNCPoint2[8052] = {X 371.5193, Y 45.9200, Z -3.0000, A 0.000, B 0.000, C 0.000 }
gfCNCPoint2[8053] = {X 388.0597, Y 45.9200, Z -3.0000, A 0.000, B 0.000, C 0.000 }
gfCNCPoint2[8054] = {X 389.4143, Y 45.9962, Z -3.0000, A 0.000, B 0.000, C 0.000 }
gfCNCPoint2[8055] = {X 390.7519, Y 46.2238, Z -3.0000, A 0.000, B 0.000, C 0.000 }
gfCNCPoint2[8056] = {X 392.0555, Y 46.6000, Z -3.0000, A 0.000, B 0.000, C 0.000 }
gfCNCPoint2[8057] = {X 393.3087, Y 47.1200, Z -3.0000, A 0.000, B 0.000, C 0.000 }
gfCNCPoint2[8058] = {X 394.2237, Y 46.7243, Z -3.0000, A 0.000, B 0.000, C 0.000 }
gfCNCPoint2[8059] = {X 395.1681, Y 46.4053, Z -3.0000, A 0.000, B 0.000, C 0.000 }
gfCNCPoint2[8060] = {X 395.0678, Y 45.7292, Z -3.0000, A 0.000, B 0.000, C 0.000 }
gfCNCPoint2[8061] = {X 395.0314, Y 45.0468, Z -3.0000, A 0.000, B 0.000, C 0.000 }
gfCNCPoint2[8062] = {X 395.0316, Y 44.1296, Z -3.0000, A 0.000, B 0.000, C 0.000 }
gfCNCPoint2[8063] = {X 395.1397, Y 42.9565, Z -3.0000, A 0.000, B 0.000, C 0.000 }
gfCNCPoint2[8064] = {X 395.4356, Y 41.8161, Z -3.0000, A 0.000, B 0.000, C 0.000 }
gfCNCPoint2[8065] = {X 395.9116, Y 40.7384, Z -3.0000, A 0.000, B 0.000, C 0.000 }
gfCNCPoint2[8066] = {X 396.5552, Y 39.7516, Z -3.0000, A 0.000, B 0.000, C 0.000 }
gfCNCPoint2[8067] = {X 396.5552, Y 32.4634, Z -3.0000, A 0.000, B 0.000, C 0.000 }
gfCNCPoint2[8068] = {X 394.6681, Y 29.1834, Z -3.0000, A 0.000, B 0.000, C 0.000 }
gfCNCPoint2[8069] = {X 396.7484, Y 27.9866, Z -3.0000, A 0.000, B 0.000, C 0.000 }
gfCNCPoint2[8070] = {X 394.7997, Y 24.5994, Z -3.0000, A 0.000, B 0.000, C 0.000 }
gfCNCPoint2[8071] = {X 393.1056, Y 21.6452, Z -3.0000, A 0.000, B 0.000, C 0.000 }
gfCNCPoint2[8072] = {X 392.1683, Y 20.0504, Z -3.0000, A 0.000, B 0.000, C 0.000 }
gfCNCPoint2[8073] = {X 391.1971, Y 18.4760, Z -3.0000, A 0.000, B 0.000, C 0.000 }
gfCNCPoint2[8074] = {X 390.8069, Y 17.9330, Z -3.0000, A 0.000, B 0.000, C 0.000 }
gfCNCPoint2[8075] = {X 390.3547, Y 17.4405, Z -3.0000, A 0.000, B 0.000, C 0.000 }
gfCNCPoint2[8076] = {X 389.5442, Y 16.9850, Z -3.0000, A 0.000, B 0.000, C 0.000 }
gfCNCPoint2[8077] = {X 388.8348, Y 16.3840, Z -3.0000, A 0.000, B 0.000, C 0.000 }
gfCNCPoint2[8078] = {X 388.2523, Y 15.6593, Z -3.0000, A 0.000, B 0.000, C 0.000 }
gfCNCPoint2[8079] = {X 387.8177, Y 14.8374, Z -3.0000, A 0.000, B 0.000, C 0.000 }
gfCNCPoint2[8080] = {X 387.5470, Y 13.9479, Z -3.0000, A 0.000, B 0.000, C 0.000 }
gfCNCPoint2[8081] = {X 387.4498, Y 13.0232, Z -3.0000, A 0.000, B 0.000, C 0.000 }
gfCNCPoint2[8082] = {X 387.4496, Y 12.1868, Z -3.0000, A 0.000, B 0.000, C 0.000 }
gfCNCPoint2[8083] = {X 387.5362, Y 11.2717, Z -3.0000, A 0.000, B 0.000, C 0.000 }
gfCNCPoint2[8084] = {X 387.7928, Y 10.3891, Z -3.0000, A 0.000, B 0.000, C 0.000 }
gfCNCPoint2[8085] = {X 388.2375, Y 9.5281, Z -3.0000, A 0.000, B 0.000, C 0.000 }
gfCNCPoint2[8086] = {X 388.8436, Y 8.7718, Z -3.0000, A 0.000, B 0.000, C 0.000 }
gfCNCPoint2[8087] = {X 389.5872, Y 8.1503, Z -3.0000, A 0.000, B 0.000, C 0.000 }
gfCNCPoint2[8088] = {X 390.4390, Y 7.6880, Z -3.0000, A 0.000, B 0.000, C 0.000 }
gfCNCPoint2[8089] = {X 391.3653, Y 7.4030, Z -3.0000, A 0.000, B 0.000, C 0.000 }
gfCNCPoint2[8090] = {X 392.3296, Y 7.3068, Z -3.0000, A 0.000, B 0.000, C 0.000 }
gfCNCPoint2[8091] = {X 399.1118, Y 7.3068, Z -3.0000, A 0.000, B 0.000, C 0.000 }
gfCNCPoint2[8092] = {X 400.0638, Y 7.4006, Z -3.0000, A 0.000, B 0.000, C 0.000 }
gfCNCPoint2[8093] = {X 400.9793, Y 7.6783, Z -3.0000, A 0.000, B 0.000, C 0.000 }
gfCNCPoint2[8094] = {X 401.8229, Y 8.1292, Z -3.0000, A 0.000, B 0.000, C 0.000 }
gfCNCPoint2[8095] = {X 402.5624, Y 8.7361, Z -3.0000, A 0.000, B 0.000, C 0.000 }
gfCNCPoint2[8096] = {X 403.1693, Y 9.4756, Z -3.0000, A 0.000, B 0.000, C 0.000 }
gfCNCPoint2[8097] = {X 403.6203, Y 10.3193, Z -3.0000, A 0.000, B 0.000, C 0.000 }
gfCNCPoint2[8098] = {X 403.8980, Y 11.2348, Z -3.0000, A 0.000, B 0.000, C 0.000 }
gfCNCPoint2[8099] = {X 403.9918, Y 12.1868, Z -3.0000, A 0.000, B 0.000, C 0.000 }
gfCNCPoint2[8100] = {X 403.9915, Y 13.0237, Z -3.0000, A 0.000, B 0.000, C 0.000 }
gfCNCPoint2[8101] = {X 403.9016, Y 13.9115, Z -3.0000, A 0.000, B 0.000, C 0.000 }
gfCNCPoint2[8102] = {X 403.6516, Y 14.7680, Z -3.0000, A 0.000, B 0.000, C 0.000 }
gfCNCPoint2[8103] = {X 405.3651, Y 17.7434, Z -3.0000, A 0.000, B 0.000, C 0.000 }
gfCNCPoint2[8104] = {X 407.2449, Y 14.6985, Z -3.0000, A 0.000, B 0.000, C 0.000 }
gfCNCPoint2[8105] = {X 407.0143, Y 13.8730, Z -3.0000, A 0.000, B 0.000, C 0.000 }
gfCNCPoint2[8106] = {X 406.9317, Y 13.0199, Z -3.0000, A 0.000, B 0.000, C 0.000 }
gfCNCPoint2[8107] = {X 406.9315, Y 12.1868, Z -3.0000, A 0.000, B 0.000, C 0.000 }
gfCNCPoint2[8108] = {X 407.0253, Y 11.2348, Z -3.0000, A 0.000, B 0.000, C 0.000 }
gfCNCPoint2[8109] = {X 407.3030, Y 10.3193, Z -3.0000, A 0.000, B 0.000, C 0.000 }
gfCNCPoint2[8110] = {X 407.7540, Y 9.4756, Z -3.0000, A 0.000, B 0.000, C 0.000 }
gfCNCPoint2[8111] = {X 408.3609, Y 8.7361, Z -3.0000, A 0.000, B 0.000, C 0.000 }
gfCNCPoint2[8112] = {X 409.1004, Y 8.1292, Z -3.0000, A 0.000, B 0.000, C 0.000 }
gfCNCPoint2[8113] = {X 409.9440, Y 7.6783, Z -3.0000, A 0.000, B 0.000, C 0.000 }
gfCNCPoint2[8114] = {X 410.8595, Y 7.4006, Z -3.0000, A 0.000, B 0.000, C 0.000 }
gfCNCPoint2[8115] = {X 411.8115, Y 7.3068, Z -3.0000, A 0.000, B 0.000, C 0.000 }
gfCNCPoint2[8116] = {X 419.3245, Y 7.3068, Z -3.0000, A 0.000, B 0.000, C 0.000 }
gfCNCPoint2[8117] = {X 420.2888, Y 7.4030, Z -3.0000, A 0.000, B 0.000, C 0.000 }
gfCNCPoint2[8118] = {X 421.2151, Y 7.6880, Z -3.0000, A 0.000, B 0.000, C 0.000 }
gfCNCPoint2[8119] = {X 422.0669, Y 8.1503, Z -3.0000, A 0.000, B 0.000, C 0.000 }
gfCNCPoint2[8120] = {X 422.8105, Y 8.7718, Z -3.0000, A 0.000, B 0.000, C 0.000 }
gfCNCPoint2[8121] = {X 423.4166, Y 9.5281, Z -3.0000, A 0.000, B 0.000, C 0.000 }
gfCNCPoint2[8122] = {X 423.8613, Y 10.3891, Z -3.0000, A 0.000, B 0.000, C 0.000 }
gfCNCPoint2[8123] = {X 424.1179, Y 11.2717, Z -3.0000, A 0.000, B 0.000, C 0.000 }
gfCNCPoint2[8124] = {X 424.2045, Y 12.1868, Z -3.0000, A 0.000, B 0.000, C 0.000 }
gfCNCPoint2[8125] = {X 424.2045, Y 12.9780, Z -3.0000, A 0.000, B 0.000, C 0.000 }
gfCNCPoint2[8126] = {X 424.1057, Y 13.9307, Z -3.0000, A 0.000, B 0.000, C 0.000 }
gfCNCPoint2[8127] = {X 423.8251, Y 14.8465, Z -3.0000, A 0.000, B 0.000, C 0.000 }
gfCNCPoint2[8128] = {X 423.3732, Y 15.6911, Z -3.0000, A 0.000, B 0.000, C 0.000 }
gfCNCPoint2[8129] = {X 422.7671, Y 16.4328, Z -3.0000, A 0.000, B 0.000, C 0.000 }
gfCNCPoint2[8130] = {X 422.0293, Y 17.0437, Z -3.0000, A 0.000, B 0.000, C 0.000 }
gfCNCPoint2[8131] = {X 421.1877, Y 17.5009, Z -3.0000, A 0.000, B 0.000, C 0.000 }
gfCNCPoint2[8132] = {X 420.5398, Y 18.3844, Z -3.0000, A 0.000, B 0.000, C 0.000 }
gfCNCPoint2[8133] = {X 419.9506, Y 19.3081, Z -3.0000, A 0.000, B 0.000, C 0.000 }
gfCNCPoint2[8134] = {X 414.1632, Y 28.6167, Z -3.0000, A 0.000, B 0.000, C 0.000 }
gfCNCPoint2[8135] = {X 422.3159, Y 33.6855, Z -3.0000, A 0.000, B 0.000, C 0.000 }
gfCNCPoint2[8136] = {X 421.8902, Y 34.3703, Z -3.0000, A 0.000, B 0.000, C 0.000 }
gfCNCPoint2[8137] = {X 422.1461, Y 34.1009, Z -3.0000, A 0.000, B 0.000, C 0.000 }
gfCNCPoint2[8138] = {X 422.4089, Y 33.8382, Z -3.0000, A 0.000, B 0.000, C 0.000 }
gfCNCPoint2[8139] = {X 422.3623, Y 33.7619, Z -3.0000, A 0.000, B 0.000, C 0.000 }
gfCNCPoint2[8140] = {X 422.3159, Y 33.6855, Z -3.0000, A 0.000, B 0.000, C 0.000 }
gfCNCPoint2[8141] = {X 420.2777, Y 32.4183, Z -3.0000, A 0.000, B 0.000, C 0.000 }
gfCNCPoint2[8142] = {X 419.3065, Y 33.9805, Z -3.0000, A 0.000, B 0.000, C 0.000 }
gfCNCPoint2[8143] = {X 419.3068, Y 38.3390, Z -3.0000, A 0.000, B 0.000, C 0.000 }
gfCNCPoint2[8144] = {X 419.9573, Y 39.7077, Z -3.0000, A 0.000, B 0.000, C 0.000 }
gfCNCPoint2[8145] = {X 420.4331, Y 41.1464, Z -3.0000, A 0.000, B 0.000, C 0.000 }
gfCNCPoint2[8146] = {X 420.6277, Y 41.1585, Z -3.0000, A 0.000, B 0.000, C 0.000 }
gfCNCPoint2[8147] = {X 420.8222, Y 41.1728, Z -3.0000, A 0.000, B 0.000, C 0.000 }
gfCNCPoint2[8148] = {X 421.2841, Y 39.7585, Z -3.0000, A 0.000, B 0.000, C 0.000 }
gfCNCPoint2[8149] = {X 421.9163, Y 38.4117, Z -3.0000, A 0.000, B 0.000, C 0.000 }
gfCNCPoint2[8150] = {X 422.7093, Y 37.1528, Z -3.0000, A 0.000, B 0.000, C 0.000 }
gfCNCPoint2[8151] = {X 423.6511, Y 36.0010, Z -3.0000, A 0.000, B 0.000, C 0.000 }
gfCNCPoint2[8152] = {X 424.3405, Y 35.3142, Z -3.0000, A 0.000, B 0.000, C 0.000 }
gfCNCPoint2[8153] = {X 425.0829, Y 34.6852, Z -3.0000, A 0.000, B 0.000, C 0.000 }
gfCNCPoint2[8154] = {X 425.4263, Y 34.0130, Z -3.0000, A 0.000, B 0.000, C 0.000 }
gfCNCPoint2[8155] = {X 424.8790, Y 33.2422, Z -3.0000, A 0.000, B 0.000, C 0.000 }
gfCNCPoint2[8156] = {X 424.3706, Y 32.4453, Z -3.0000, A 0.000, B 0.000, C 0.000 }
gfCNCPoint2[8157] = {X 423.3898, Y 30.5987, Z -3.0000, A 0.000, B 0.000, C 0.000 }
gfCNCPoint2[8158] = {X 422.6169, Y 28.6559, Z -3.0000, A 0.000, B 0.000, C 0.000 }
gfCNCPoint2[8159] = {X 420.2777, Y 32.4183, Z -3.0000, A 0.000, B 0.000, C 0.000 }
gfCNCPoint2[8160] = {X 418.2395, Y 31.1511, Z -3.0000, A 0.000, B 0.000, C 0.000 }
gfCNCPoint2[8161] = {X 416.9064, Y 33.2954, Z -3.0000, A 0.000, B 0.000, C 0.000 }
gfCNCPoint2[8162] = {X 416.9068, Y 38.9957, Z -3.0000, A 0.000, B 0.000, C 0.000 }
gfCNCPoint2[8163] = {X 417.4882, Y 40.0489, Z -3.0000, A 0.000, B 0.000, C 0.000 }
gfCNCPoint2[8164] = {X 417.9363, Y 41.1653, Z -3.0000, A 0.000, B 0.000, C 0.000 }
gfCNCPoint2[8165] = {X 418.2443, Y 42.3282, Z -3.0000, A 0.000, B 0.000, C 0.000 }
gfCNCPoint2[8166] = {X 418.4075, Y 43.5200, Z -3.0000, A 0.000, B 0.000, C 0.000 }
gfCNCPoint2[8167] = {X 419.4886, Y 43.5200, Z -3.0000, A 0.000, B 0.000, C 0.000 }
gfCNCPoint2[8168] = {X 421.1752, Y 43.6186, Z -3.0000, A 0.000, B 0.000, C 0.000 }
gfCNCPoint2[8169] = {X 422.8389, Y 43.9129, Z -3.0000, A 0.000, B 0.000, C 0.000 }
gfCNCPoint2[8170] = {X 423.0005, Y 42.4234, Z -3.0000, A 0.000, B 0.000, C 0.000 }
gfCNCPoint2[8171] = {X 423.3900, Y 40.9766, Z -3.0000, A 0.000, B 0.000, C 0.000 }
gfCNCPoint2[8172] = {X 423.9980, Y 39.6073, Z -3.0000, A 0.000, B 0.000, C 0.000 }
gfCNCPoint2[8173] = {X 424.8102, Y 38.3482, Z -3.0000, A 0.000, B 0.000, C 0.000 }
gfCNCPoint2[8174] = {X 425.8068, Y 37.2295, Z -3.0000, A 0.000, B 0.000, C 0.000 }
gfCNCPoint2[8175] = {X 426.9642, Y 36.2780, Z -3.0000, A 0.000, B 0.000, C 0.000 }
gfCNCPoint2[8176] = {X 428.2765, Y 33.7094, Z -3.0000, A 0.000, B 0.000, C 0.000 }
gfCNCPoint2[8177] = {X 427.2127, Y 32.3918, Z -3.0000, A 0.000, B 0.000, C 0.000 }
gfCNCPoint2[8178] = {X 426.2879, Y 30.9732, Z -3.0000, A 0.000, B 0.000, C 0.000 }
gfCNCPoint2[8179] = {X 425.5118, Y 29.4682, Z -3.0000, A 0.000, B 0.000, C 0.000 }
gfCNCPoint2[8180] = {X 424.8922, Y 27.8923, Z -3.0000, A 0.000, B 0.000, C 0.000 }
gfCNCPoint2[8181] = {X 424.8104, Y 27.6418, Z -3.0000, A 0.000, B 0.000, C 0.000 }
gfCNCPoint2[8182] = {X 424.7325, Y 27.3900, Z -3.0000, A 0.000, B 0.000, C 0.000 }
gfCNCPoint2[8183] = {X 424.2998, Y 25.6528, Z -3.0000, A 0.000, B 0.000, C 0.000 }
gfCNCPoint2[8184] = {X 424.0103, Y 23.8860, Z -3.0000, A 0.000, B 0.000, C 0.000 }
gfCNCPoint2[8185] = {X 423.8659, Y 22.1015, Z -3.0000, A 0.000, B 0.000, C 0.000 }
gfCNCPoint2[8186] = {X 418.2395, Y 31.1511, Z -3.0000, A 0.000, B 0.000, C 0.000 }
gfCNCPoint2[8187] = {X 416.2013, Y 29.8839, Z -3.0000, A 0.000, B 0.000, C 0.000 }
gfCNCPoint2[8188] = {X 414.5064, Y 32.6102, Z -3.0000, A 0.000, B 0.000, C 0.000 }
gfCNCPoint2[8189] = {X 414.5069, Y 39.7472, Z -3.0000, A 0.000, B 0.000, C 0.000 }
gfCNCPoint2[8190] = {X 415.1555, Y 40.7521, Z -3.0000, A 0.000, B 0.000, C 0.000 }
gfCNCPoint2[8191] = {X 415.6338, Y 41.8482, Z -3.0000, A 0.000, B 0.000, C 0.000 }
gfCNCPoint2[8192] = {X 415.9295, Y 43.0071, Z -3.0000, A 0.000, B 0.000, C 0.000 }
gfCNCPoint2[8193] = {X 416.0347, Y 44.1985, Z -3.0000, A 0.000, B 0.000, C 0.000 }
gfCNCPoint2[8194] = {X 416.0347, Y 44.9999, Z -3.0000, A 0.000, B 0.000, C 0.000 }
gfCNCPoint2[8195] = {X 416.0201, Y 45.4609, Z -3.0000, A 0.000, B 0.000, C 0.000 }
gfCNCPoint2[8196] = {X 415.9763, Y 45.9200, Z -3.0000, A 0.000, B 0.000, C 0.000 }
gfCNCPoint2[8197] = {X 419.4886, Y 45.9200, Z -3.0000, A 0.000, B 0.000, C 0.000 }
gfCNCPoint2[8198] = {X 420.8957, Y 46.0022, Z -3.0000, A 0.000, B 0.000, C 0.000 }
gfCNCPoint2[8199] = {X 422.2836, Y 46.2478, Z -3.0000, A 0.000, B 0.000, C 0.000 }
gfCNCPoint2[8200] = {X 423.4822, Y 46.5992, Z -3.0000, A 0.000, B 0.000, C 0.000 }
gfCNCPoint2[8201] = {X 424.6380, Y 47.0725, Z -3.0000, A 0.000, B 0.000, C 0.000 }
gfCNCPoint2[8202] = {X 425.7388, Y 47.6626, Z -3.0000, A 0.000, B 0.000, C 0.000 }
gfCNCPoint2[8203] = {X 425.4600, Y 46.7984, Z -3.0000, A 0.000, B 0.000, C 0.000 }
gfCNCPoint2[8204] = {X 425.2910, Y 45.9063, Z -3.0000, A 0.000, B 0.000, C 0.000 }
gfCNCPoint2[8205] = {X 425.2344, Y 45.0000, Z -3.0000, A 0.000, B 0.000, C 0.000 }
gfCNCPoint2[8206] = {X 425.2344, Y 44.2090, Z -3.0000, A 0.000, B 0.000, C 0.000 }
gfCNCPoint2[8207] = {X 425.2353, Y 44.0976, Z -3.0000, A 0.000, B 0.000, C 0.000 }
gfCNCPoint2[8208] = {X 425.2378, Y 43.9863, Z -3.0000, A 0.000, B 0.000, C 0.000 }
gfCNCPoint2[8209] = {X 425.3770, Y 42.7748, Z -3.0000, A 0.000, B 0.000, C 0.000 }
gfCNCPoint2[8210] = {X 425.7165, Y 41.6036, Z -3.0000, A 0.000, B 0.000, C 0.000 }
gfCNCPoint2[8211] = {X 426.2468, Y 40.5054, Z -3.0000, A 0.000, B 0.000, C 0.000 }
gfCNCPoint2[8212] = {X 426.9528, Y 39.5112, Z -3.0000, A 0.000, B 0.000, C 0.000 }
gfCNCPoint2[8213] = {X 427.8150, Y 38.6488, Z -3.0000, A 0.000, B 0.000, C 0.000 }
gfCNCPoint2[8214] = {X 428.8090, Y 37.9424, Z -3.0000, A 0.000, B 0.000, C 0.000 }
gfCNCPoint2[8215] = {X 431.2070, Y 33.2484, Z -3.0000, A 0.000, B 0.000, C 0.000 }
gfCNCPoint2[8216] = {X 430.0933, Y 32.1405, Z -3.0000, A 0.000, B 0.000, C 0.000 }
gfCNCPoint2[8217] = {X 429.1080, Y 30.9171, Z -3.0000, A 0.000, B 0.000, C 0.000 }
gfCNCPoint2[8218] = {X 428.2631, Y 29.5928, Z -3.0000, A 0.000, B 0.000, C 0.000 }
gfCNCPoint2[8219] = {X 427.5687, Y 28.1837, Z -3.0000, A 0.000, B 0.000, C 0.000 }
gfCNCPoint2[8220] = {X 427.0332, Y 26.7069, Z -3.0000, A 0.000, B 0.000, C 0.000 }
gfCNCPoint2[8221] = {X 426.6492, Y 25.1625, Z -3.0000, A 0.000, B 0.000, C 0.000 }
gfCNCPoint2[8222] = {X 426.3923, Y 23.5919, Z -3.0000, A 0.000, B 0.000, C 0.000 }
gfCNCPoint2[8223] = {X 426.2640, Y 22.0057, Z -3.0000, A 0.000, B 0.000, C 0.000 }
gfCNCPoint2[8224] = {X 426.2907, Y 19.9398, Z -3.0000, A 0.000, B 0.000, C 0.000 }
gfCNCPoint2[8225] = {X 426.5355, Y 17.8883, Z -3.0000, A 0.000, B 0.000, C 0.000 }
gfCNCPoint2[8226] = {X 426.9956, Y 15.8741, Z -3.0000, A 0.000, B 0.000, C 0.000 }
gfCNCPoint2[8227] = {X 427.6131, Y 14.1182, Z -3.0000, A 0.000, B 0.000, C 0.000 }
gfCNCPoint2[8228] = {X 428.4468, Y 12.4541, Z -3.0000, A 0.000, B 0.000, C 0.000 }
gfCNCPoint2[8229] = {X 429.4834, Y 10.9082, Z -3.0000, A 0.000, B 0.000, C 0.000 }
gfCNCPoint2[8230] = {X 430.7064, Y 9.5050, Z -3.0000, A 0.000, B 0.000, C 0.000 }
gfCNCPoint2[8231] = {X 426.0925, Y 9.5050, Z -3.0000, A 0.000, B 0.000, C 0.000 }
gfCNCPoint2[8232] = {X 426.3754, Y 10.3751, Z -3.0000, A 0.000, B 0.000, C 0.000 }
gfCNCPoint2[8233] = {X 426.5470, Y 11.2737, Z -3.0000, A 0.000, B 0.000, C 0.000 }
gfCNCPoint2[8234] = {X 426.6045, Y 12.1868, Z -3.0000, A 0.000, B 0.000, C 0.000 }
gfCNCPoint2[8235] = {X 426.6045, Y 12.9856, Z -3.0000, A 0.000, B 0.000, C 0.000 }
gfCNCPoint2[8236] = {X 426.4812, Y 14.2873, Z -3.0000, A 0.000, B 0.000, C 0.000 }
gfCNCPoint2[8237] = {X 426.1291, Y 15.5466, Z -3.0000, A 0.000, B 0.000, C 0.000 }
gfCNCPoint2[8238] = {X 425.5592, Y 16.7235, Z -3.0000, A 0.000, B 0.000, C 0.000 }
gfCNCPoint2[8239] = {X 424.7898, Y 17.7808, Z -3.0000, A 0.000, B 0.000, C 0.000 }
gfCNCPoint2[8240] = {X 423.8451, Y 18.6849, Z -3.0000, A 0.000, B 0.000, C 0.000 }
gfCNCPoint2[8241] = {X 422.7551, Y 19.4071, Z -3.0000, A 0.000, B 0.000, C 0.000 }
gfCNCPoint2[8242] = {X 422.3650, Y 19.9716, Z -3.0000, A 0.000, B 0.000, C 0.000 }
gfCNCPoint2[8243] = {X 422.0020, Y 20.5540, Z -3.0000, A 0.000, B 0.000, C 0.000 }
gfCNCPoint2[8244] = {X 416.2013, Y 29.8839, Z -3.0000, A 0.000, B 0.000, C 0.000 }
gfCNCPoint2[8245] = {X 414.1632, Y 28.6167, Z -3.0000, A 0.000, B 0.000, C 0.000 }
gfCNCPoint2[8246] = {X 412.1063, Y 31.9250, Z -3.0000, A 0.000, B 0.000, C 0.000 }
gfCNCPoint2[8247] = {X 412.1070, Y 40.6521, Z -3.0000, A 0.000, B 0.000, C 0.000 }
gfCNCPoint2[8248] = {X 412.7487, Y 41.4086, Z -3.0000, A 0.000, B 0.000, C 0.000 }
gfCNCPoint2[8249] = {X 413.2286, Y 42.2768, Z -3.0000, A 0.000, B 0.000, C 0.000 }
gfCNCPoint2[8250] = {X 413.5278, Y 43.2226, Z -3.0000, A 0.000, B 0.000, C 0.000 }
gfCNCPoint2[8251] = {X 413.6347, Y 44.2089, Z -3.0000, A 0.000, B 0.000, C 0.000 }
gfCNCPoint2[8252] = {X 413.6347, Y 45.0000, Z -3.0000, A 0.000, B 0.000, C 0.000 }
gfCNCPoint2[8253] = {X 413.6249, Y 45.3090, Z -3.0000, A 0.000, B 0.000, C 0.000 }
gfCNCPoint2[8254] = {X 413.5956, Y 45.6167, Z -3.0000, A 0.000, B 0.000, C 0.000 }
gfCNCPoint2[8255] = {X 413.3652, Y 46.5992, Z -3.0000, A 0.000, B 0.000, C 0.000 }
gfCNCPoint2[8256] = {X 412.9377, Y 47.5134, Z -3.0000, A 0.000, B 0.000, C 0.000 }
gfCNCPoint2[8257] = {X 412.3313, Y 48.3200, Z -3.0000, A 0.000, B 0.000, C 0.000 }
gfCNCPoint2[8258] = {X 411.9795, Y 47.9934, Z -3.0000, A 0.000, B 0.000, C 0.000 }
gfCNCPoint2[8259] = {X 411.3003, Y 48.5889, Z -3.0000, A 0.000, B 0.000, C 0.000 }
gfCNCPoint2[8260] = {X 410.5138, Y 49.0331, Z -3.0000, A 0.000, B 0.000, C 0.000 }
gfCNCPoint2[8261] = {X 409.6532, Y 49.3073, Z -3.0000, A 0.000, B 0.000, C 0.000 }
gfCNCPoint2[8262] = {X 408.7547, Y 49.4000, Z -3.0000, A 0.000, B 0.000, C 0.000 }
gfCNCPoint2[8263] = {X 402.3112, Y 49.4000, Z -3.0000, A 0.000, B 0.000, C 0.000 }
gfCNCPoint2[8264] = {X 401.3321, Y 49.2897, Z -3.0000, A 0.000, B 0.000, C 0.000 }
gfCNCPoint2[8265] = {X 400.4021, Y 48.9643, Z -3.0000, A 0.000, B 0.000, C 0.000 }
gfCNCPoint2[8266] = {X 399.5678, Y 48.4400, Z -3.0000, A 0.000, B 0.000, C 0.000 }
gfCNCPoint2[8267] = {X 398.8711, Y 47.7433, Z -3.0000, A 0.000, B 0.000, C 0.000 }
gfCNCPoint2[8268] = {X 398.3469, Y 46.9091, Z -3.0000, A 0.000, B 0.000, C 0.000 }
gfCNCPoint2[8269] = {X 398.0215, Y 45.9791, Z -3.0000, A 0.000, B 0.000, C 0.000 }
gfCNCPoint2[8270] = {X 397.9112, Y 45.0000, Z -3.0000, A 0.000, B 0.000, C 0.000 }
gfCNCPoint2[8271] = {X 397.9116, Y 44.1518, Z -3.0000, A 0.000, B 0.000, C 0.000 }
gfCNCPoint2[8272] = {X 398.0215, Y 43.2300, Z -3.0000, A 0.000, B 0.000, C 0.000 }
gfCNCPoint2[8273] = {X 398.3223, Y 42.3519, Z -3.0000, A 0.000, B 0.000, C 0.000 }
gfCNCPoint2[8274] = {X 398.8006, Y 41.5563, Z -3.0000, A 0.000, B 0.000, C 0.000 }
gfCNCPoint2[8275] = {X 399.4352, Y 40.8789, Z -3.0000, A 0.000, B 0.000, C 0.000 }
gfCNCPoint2[8276] = {X 399.4352, Y 31.6940, Z -3.0000, A 0.000, B 0.000, C 0.000 }
gfCNCPoint2[8277] = {X 395.2158, Y 24.3600, Z -3.0000, A 0.000, B 0.000, C 0.000 }
gfCNCPoint2[8278] = {X 393.5220, Y 21.4064, Z -3.0000, A 0.000, B 0.000, C 0.000 }
gfCNCPoint2[8279] = {X 392.5795, Y 19.8028, Z -3.0000, A 0.000, B 0.000, C 0.000 }
gfCNCPoint2[8280] = {X 391.6029, Y 18.2196, Z -3.0000, A 0.000, B 0.000, C 0.000 }
gfCNCPoint2[8281] = {X 391.1509, Y 17.5956, Z -3.0000, A 0.000, B 0.000, C 0.000 }
gfCNCPoint2[8282] = {X 390.6236, Y 17.0338, Z -3.0000, A 0.000, B 0.000, C 0.000 }
gfCNCPoint2[8283] = {X 389.8685, Y 16.6253, Z -3.0000, A 0.000, B 0.000, C 0.000 }
gfCNCPoint2[8284] = {X 389.2070, Y 16.0779, Z -3.0000, A 0.000, B 0.000, C 0.000 }
gfCNCPoint2[8285] = {X 388.6645, Y 15.4125, Z -3.0000, A 0.000, B 0.000, C 0.000 }
gfCNCPoint2[8286] = {X 388.2615, Y 14.6544, Z -3.0000, A 0.000, B 0.000, C 0.000 }
gfCNCPoint2[8287] = {X 388.0134, Y 13.8324, Z -3.0000, A 0.000, B 0.000, C 0.000 }
gfCNCPoint2[8288] = {X 387.9296, Y 12.9779, Z -3.0000, A 0.000, B 0.000, C 0.000 }
gfCNCPoint2[8289] = {X 387.9296, Y 12.1868, Z -3.0000, A 0.000, B 0.000, C 0.000 }
gfCNCPoint2[8290] = {X 388.0399, Y 11.2077, Z -3.0000, A 0.000, B 0.000, C 0.000 }
gfCNCPoint2[8291] = {X 388.3654, Y 10.2777, Z -3.0000, A 0.000, B 0.000, C 0.000 }
gfCNCPoint2[8292] = {X 388.8896, Y 9.4435, Z -3.0000, A 0.000, B 0.000, C 0.000 }
gfCNCPoint2[8293] = {X 389.5863, Y 8.7468, Z -3.0000, A 0.000, B 0.000, C 0.000 }
gfCNCPoint2[8294] = {X 390.4205, Y 8.2226, Z -3.0000, A 0.000, B 0.000, C 0.000 }
gfCNCPoint2[8295] = {X 391.3505, Y 7.8971, Z -3.0000, A 0.000, B 0.000, C 0.000 }
gfCNCPoint2[8296] = {X 392.3296, Y 7.7868, Z -3.0000, A 0.000, B 0.000, C 0.000 }
gfCNCPoint2[8297] = {X 399.1118, Y 7.7868, Z -3.0000, A 0.000, B 0.000, C 0.000 }
gfCNCPoint2[8298] = {X 400.0909, Y 7.8971, Z -3.0000, A 0.000, B 0.000, C 0.000 }
gfCNCPoint2[8299] = {X 401.0208, Y 8.2226, Z -3.0000, A 0.000, B 0.000, C 0.000 }
gfCNCPoint2[8300] = {X 401.8551, Y 8.7468, Z -3.0000, A 0.000, B 0.000, C 0.000 }
gfCNCPoint2[8301] = {X 402.5518, Y 9.4435, Z -3.0000, A 0.000, B 0.000, C 0.000 }
gfCNCPoint2[8302] = {X 403.0760, Y 10.2777, Z -3.0000, A 0.000, B 0.000, C 0.000 }
gfCNCPoint2[8303] = {X 403.4014, Y 11.2077, Z -3.0000, A 0.000, B 0.000, C 0.000 }
gfCNCPoint2[8304] = {X 403.5118, Y 12.1868, Z -3.0000, A 0.000, B 0.000, C 0.000 }
gfCNCPoint2[8305] = {X 403.5115, Y 13.0233, Z -3.0000, A 0.000, B 0.000, C 0.000 }
gfCNCPoint2[8306] = {X 403.4070, Y 13.9326, Z -3.0000, A 0.000, B 0.000, C 0.000 }
gfCNCPoint2[8307] = {X 403.1165, Y 14.8007, Z -3.0000, A 0.000, B 0.000, C 0.000 }
gfCNCPoint2[8308] = {X 405.3508, Y 18.6803, Z -3.0000, A 0.000, B 0.000, C 0.000 }
gfCNCPoint2[8309] = {X 407.7812, Y 14.7434, Z -3.0000, A 0.000, B 0.000, C 0.000 }
gfCNCPoint2[8310] = {X 407.5049, Y 13.8798, Z -3.0000, A 0.000, B 0.000, C 0.000 }
gfCNCPoint2[8311] = {X 407.4115, Y 12.9779, Z -3.0000, A 0.000, B 0.000, C 0.000 }
gfCNCPoint2[8312] = {X 407.4115, Y 12.1868, Z -3.0000, A 0.000, B 0.000, C 0.000 }
gfCNCPoint2[8313] = {X 407.5219, Y 11.2077, Z -3.0000, A 0.000, B 0.000, C 0.000 }
gfCNCPoint2[8314] = {X 407.8473, Y 10.2777, Z -3.0000, A 0.000, B 0.000, C 0.000 }
gfCNCPoint2[8315] = {X 408.3715, Y 9.4435, Z -3.0000, A 0.000, B 0.000, C 0.000 }
gfCNCPoint2[8316] = {X 409.0682, Y 8.7468, Z -3.0000, A 0.000, B 0.000, C 0.000 }
gfCNCPoint2[8317] = {X 409.9025, Y 8.2226, Z -3.0000, A 0.000, B 0.000, C 0.000 }
gfCNCPoint2[8318] = {X 410.8324, Y 7.8971, Z -3.0000, A 0.000, B 0.000, C 0.000 }
gfCNCPoint2[8319] = {X 411.8115, Y 7.7868, Z -3.0000, A 0.000, B 0.000, C 0.000 }
gfCNCPoint2[8320] = {X 419.3245, Y 7.7868, Z -3.0000, A 0.000, B 0.000, C 0.000 }
gfCNCPoint2[8321] = {X 420.3036, Y 7.8971, Z -3.0000, A 0.000, B 0.000, C 0.000 }
gfCNCPoint2[8322] = {X 421.2335, Y 8.2226, Z -3.0000, A 0.000, B 0.000, C 0.000 }
gfCNCPoint2[8323] = {X 422.0678, Y 8.7468, Z -3.0000, A 0.000, B 0.000, C 0.000 }
gfCNCPoint2[8324] = {X 422.7645, Y 9.4435, Z -3.0000, A 0.000, B 0.000, C 0.000 }
gfCNCPoint2[8325] = {X 423.2887, Y 10.2777, Z -3.0000, A 0.000, B 0.000, C 0.000 }
gfCNCPoint2[8326] = {X 423.6141, Y 11.2077, Z -3.0000, A 0.000, B 0.000, C 0.000 }
gfCNCPoint2[8327] = {X 423.7245, Y 12.1868, Z -3.0000, A 0.000, B 0.000, C 0.000 }
gfCNCPoint2[8328] = {X 423.7244, Y 12.9810, Z -3.0000, A 0.000, B 0.000, C 0.000 }
gfCNCPoint2[8329] = {X 423.6302, Y 13.8598, Z -3.0000, A 0.000, B 0.000, C 0.000 }
gfCNCPoint2[8330] = {X 423.3648, Y 14.7028, Z -3.0000, A 0.000, B 0.000, C 0.000 }
gfCNCPoint2[8331] = {X 422.9386, Y 15.4770, Z -3.0000, A 0.000, B 0.000, C 0.000 }
gfCNCPoint2[8332] = {X 422.3683, Y 16.1521, Z -3.0000, A 0.000, B 0.000, C 0.000 }
gfCNCPoint2[8333] = {X 421.6761, Y 16.7017, Z -3.0000, A 0.000, B 0.000, C 0.000 }
gfCNCPoint2[8334] = {X 420.8894, Y 17.1043, Z -3.0000, A 0.000, B 0.000, C 0.000 }
gfCNCPoint2[8335] = {X 420.1824, Y 18.0570, Z -3.0000, A 0.000, B 0.000, C 0.000 }
gfCNCPoint2[8336] = {X 419.5422, Y 19.0559, Z -3.0000, A 0.000, B 0.000, C 0.000 }
gfCNCPoint2[8337] = {X 418.0618, Y 21.4531, Z -3.0000, A 0.000, B 0.000, C 0.000 }
gfCNCPoint2[8338] = {X 411.6263, Y 31.7878, Z -3.0000, A 0.000, B 0.000, C 0.000 }
gfCNCPoint2[8339] = {X 411.6270, Y 40.8620, Z -3.0000, A 0.000, B 0.000, C 0.000 }
gfCNCPoint2[8340] = {X 412.2660, Y 41.5588, Z -3.0000, A 0.000, B 0.000, C 0.000 }
gfCNCPoint2[8341] = {X 412.7463, Y 42.3732, Z -3.0000, A 0.000, B 0.000, C 0.000 }
gfCNCPoint2[8342] = {X 413.0469, Y 43.2696, Z -3.0000, A 0.000, B 0.000, C 0.000 }
gfCNCPoint2[8343] = {X 413.1547, Y 44.2089, Z -3.0000, A 0.000, B 0.000, C 0.000 }
gfCNCPoint2[8344] = {X 413.1545, Y 45.0423, Z -3.0000, A 0.000, B 0.000, C 0.000 }
gfCNCPoint2[8345] = {X 413.0719, Y 45.8494, Z -3.0000, A 0.000, B 0.000, C 0.000 }
gfCNCPoint2[8346] = {X 412.8426, Y 46.6276, Z -3.0000, A 0.000, B 0.000, C 0.000 }
gfCNCPoint2[8347] = {X 412.4743, Y 47.3505, Z -3.0000, A 0.000, B 0.000, C 0.000 }
gfCNCPoint2[8348] = {X 411.9795, Y 47.9934, Z -3.0000, A 0.000, B 0.000, C 0.000 }
gfCNCPoint2[8349] = {X 412.3313, Y 48.3200, Z -3.0000, A 0.000, B 0.000, C 0.000 }
gfCNCPoint2[8350] = {X 419.4886, Y 48.3200, Z -3.0000, A 0.000, B 0.000, C 0.000 }
gfCNCPoint2[8351] = {X 420.8006, Y 48.4093, Z -3.0000, A 0.000, B 0.000, C 0.000 }
gfCNCPoint2[8352] = {X 422.0883, Y 48.6756, Z -3.0000, A 0.000, B 0.000, C 0.000 }
gfCNCPoint2[8353] = {X 423.3281, Y 49.1140, Z -3.0000, A 0.000, B 0.000, C 0.000 }
gfCNCPoint2[8354] = {X 424.4970, Y 49.7164, Z -3.0000, A 0.000, B 0.000, C 0.000 }
gfCNCPoint2[8355] = {X 425.4625, Y 50.3832, Z -3.0000, A 0.000, B 0.000, C 0.000 }
gfCNCPoint2[8356] = {X 426.3402, Y 51.1620, Z -3.0000, A 0.000, B 0.000, C 0.000 }
gfCNCPoint2[8357] = {X 427.1172, Y 52.0412, Z -3.0000, A 0.000, B 0.000, C 0.000 }
gfCNCPoint2[8358] = {X 427.7821, Y 53.0080, Z -3.0000, A 0.000, B 0.000, C 0.000 }
gfCNCPoint2[8359] = {X 428.1269, Y 53.6316, Z -3.0000, A 0.000, B 0.000, C 0.000 }
gfCNCPoint2[8360] = {X 428.4248, Y 54.2789, Z -3.0000, A 0.000, B 0.000, C 0.000 }
gfCNCPoint2[8361] = {X 431.5823, Y 55.5095, Z -3.0000, A 0.000, B 0.000, C 0.000 }
gfCNCPoint2[8362] = {X 439.8774, Y 58.8005, Z -3.0000, A 0.000, B 0.000, C 0.000 }
gfCNCPoint2[8363] = {X 441.6476, Y 54.3389, Z -3.0000, A 0.000, B 0.000, C 0.000 }
gfCNCPoint2[8364] = {X 444.2222, Y 55.3604, Z -3.0000, A 0.000, B 0.000, C 0.000 }
gfCNCPoint2[8365] = {X 444.5425, Y 54.0019, Z -3.0000, A 0.000, B 0.000, C 0.000 }
gfCNCPoint2[8366] = {X 444.9921, Y 52.6806, Z -3.0000, A 0.000, B 0.000, C 0.000 }
gfCNCPoint2[8367] = {X 443.9521, Y 53.3764, Z -3.0000, A 0.000, B 0.000, C 0.000 }
gfCNCPoint2[8368] = {X 442.8310, Y 53.9323, Z -3.0000, A 0.000, B 0.000, C 0.000 }
gfCNCPoint2[8369] = {X 441.6476, Y 54.3389, Z -3.0000, A 0.000, B 0.000, C 0.000 }
gfCNCPoint2[8370] = {X 440.7625, Y 56.5697, Z -3.0000, A 0.000, B 0.000, C 0.000 }
gfCNCPoint2[8371] = {X 446.3797, Y 58.7984, Z -3.0000, A 0.000, B 0.000, C 0.000 }
gfCNCPoint2[8372] = {X 446.3796, Y 58.0000, Z -3.0000, A 0.000, B 0.000, C 0.000 }
gfCNCPoint2[8373] = {X 446.4303, Y 56.8943, Z -3.0000, A 0.000, B 0.000, C 0.000 }
gfCNCPoint2[8374] = {X 446.5820, Y 55.7979, Z -3.0000, A 0.000, B 0.000, C 0.000 }
gfCNCPoint2[8375] = {X 446.8492, Y 54.6646, Z -3.0000, A 0.000, B 0.000, C 0.000 }
gfCNCPoint2[8376] = {X 447.2243, Y 53.5622, Z -3.0000, A 0.000, B 0.000, C 0.000 }
gfCNCPoint2[8377] = {X 447.8767, Y 52.1752, Z -3.0000, A 0.000, B 0.000, C 0.000 }
gfCNCPoint2[8378] = {X 448.6995, Y 50.8820, Z -3.0000, A 0.000, B 0.000, C 0.000 }
gfCNCPoint2[8379] = {X 447.8224, Y 50.1272, Z -3.0000, A 0.000, B 0.000, C 0.000 }
gfCNCPoint2[8380] = {X 447.0760, Y 49.2431, Z -3.0000, A 0.000, B 0.000, C 0.000 }
gfCNCPoint2[8381] = {X 446.4792, Y 48.2518, Z -3.0000, A 0.000, B 0.000, C 0.000 }
gfCNCPoint2[8382] = {X 446.0469, Y 47.1785, Z -3.0000, A 0.000, B 0.000, C 0.000 }
gfCNCPoint2[8383] = {X 445.6333, Y 48.2126, Z -3.0000, A 0.000, B 0.000, C 0.000 }
gfCNCPoint2[8384] = {X 445.0668, Y 49.1715, Z -3.0000, A 0.000, B 0.000, C 0.000 }
gfCNCPoint2[8385] = {X 444.3606, Y 50.0328, Z -3.0000, A 0.000, B 0.000, C 0.000 }
gfCNCPoint2[8386] = {X 443.5314, Y 50.7763, Z -3.0000, A 0.000, B 0.000, C 0.000 }
gfCNCPoint2[8387] = {X 442.7492, Y 51.2996, Z -3.0000, A 0.000, B 0.000, C 0.000 }
gfCNCPoint2[8388] = {X 441.9061, Y 51.7177, Z -3.0000, A 0.000, B 0.000, C 0.000 }
gfCNCPoint2[8389] = {X 441.0161, Y 52.0235, Z -3.0000, A 0.000, B 0.000, C 0.000 }
gfCNCPoint2[8390] = {X 440.0668, Y 52.2156, Z -3.0000, A 0.000, B 0.000, C 0.000 }
gfCNCPoint2[8391] = {X 439.1005, Y 52.2800, Z -3.0000, A 0.000, B 0.000, C 0.000 }
gfCNCPoint2[8392] = {X 432.5144, Y 52.2800, Z -3.0000, A 0.000, B 0.000, C 0.000 }
gfCNCPoint2[8393] = {X 431.6034, Y 52.2228, Z -3.0000, A 0.000, B 0.000, C 0.000 }
gfCNCPoint2[8394] = {X 430.7067, Y 52.0520, Z -3.0000, A 0.000, B 0.000, C 0.000 }
gfCNCPoint2[8395] = {X 429.8384, Y 51.7703, Z -3.0000, A 0.000, B 0.000, C 0.000 }
gfCNCPoint2[8396] = {X 430.0171, Y 52.0775, Z -3.0000, A 0.000, B 0.000, C 0.000 }
gfCNCPoint2[8397] = {X 430.1868, Y 52.3897, Z -3.0000, A 0.000, B 0.000, C 0.000 }
gfCNCPoint2[8398] = {X 432.4640, Y 53.2773, Z -3.0000, A 0.000, B 0.000, C 0.000 }
gfCNCPoint2[8399] = {X 440.7625, Y 56.5697, Z -3.0000, A 0.000, B 0.000, C 0.000 }
gfCNCPoint2[8400] = {X 439.8774, Y 58.8005, Z -3.0000, A 0.000, B 0.000, C 0.000 }
gfCNCPoint2[8401] = {X 449.5097, Y 62.6222, Z -3.0000, A 0.000, B 0.000, C 0.000 }
gfCNCPoint2[8402] = {X 449.1115, Y 61.4471, Z -3.0000, A 0.000, B 0.000, C 0.000 }
gfCNCPoint2[8403] = {X 448.8668, Y 60.2307, Z -3.0000, A 0.000, B 0.000, C 0.000 }
gfCNCPoint2[8404] = {X 448.7798, Y 58.9930, Z -3.0000, A 0.000, B 0.000, C 0.000 }
gfCNCPoint2[8405] = {X 448.7796, Y 58.0000, Z -3.0000, A 0.000, B 0.000, C 0.000 }
gfCNCPoint2[8406] = {X 448.8564, Y 56.7833, Z -3.0000, A 0.000, B 0.000, C 0.000 }
gfCNCPoint2[8407] = {X 449.0855, Y 55.5859, Z -3.0000, A 0.000, B 0.000, C 0.000 }
gfCNCPoint2[8408] = {X 449.4632, Y 54.4268, Z -3.0000, A 0.000, B 0.000, C 0.000 }
gfCNCPoint2[8409] = {X 449.9837, Y 53.3244, Z -3.0000, A 0.000, B 0.000, C 0.000 }
gfCNCPoint2[8410] = {X 450.6386, Y 52.2961, Z -3.0000, A 0.000, B 0.000, C 0.000 }
gfCNCPoint2[8411] = {X 451.3887, Y 51.3890, Z -3.0000, A 0.000, B 0.000, C 0.000 }
gfCNCPoint2[8412] = {X 452.2434, Y 50.5796, Z -3.0000, A 0.000, B 0.000, C 0.000 }
gfCNCPoint2[8413] = {X 453.1901, Y 49.8800, Z -3.0000, A 0.000, B 0.000, C 0.000 }
gfCNCPoint2[8414] = {X 452.3731, Y 49.8442, Z -3.0000, A 0.000, B 0.000, C 0.000 }
gfCNCPoint2[8415] = {X 451.5735, Y 49.6724, Z -3.0000, A 0.000, B 0.000, C 0.000 }
gfCNCPoint2[8416] = {X 450.8138, Y 49.3696, Z -3.0000, A 0.000, B 0.000, C 0.000 }
gfCNCPoint2[8417] = {X 450.1154, Y 48.9441, Z -3.0000, A 0.000, B 0.000, C 0.000 }
gfCNCPoint2[8418] = {X 449.3503, Y 48.2496, Z -3.0000, A 0.000, B 0.000, C 0.000 }
gfCNCPoint2[8419] = {X 448.7486, Y 47.4095, Z -3.0000, A 0.000, B 0.000, C 0.000 }
gfCNCPoint2[8420] = {X 448.3373, Y 46.4616, Z -3.0000, A 0.000, B 0.000, C 0.000 }
gfCNCPoint2[8421] = {X 448.1732, Y 45.7588, Z -3.0000, A 0.000, B 0.000, C 0.000 }
gfCNCPoint2[8422] = {X 448.1146, Y 45.0395, Z -3.0000, A 0.000, B 0.000, C 0.000 }
gfCNCPoint2[8423] = {X 448.1149, Y 44.1417, Z -3.0000, A 0.000, B 0.000, C 0.000 }
gfCNCPoint2[8424] = {X 448.2252, Y 43.1751, Z -3.0000, A 0.000, B 0.000, C 0.000 }
gfCNCPoint2[8425] = {X 448.5250, Y 42.2497, Z -3.0000, A 0.000, B 0.000, C 0.000 }
gfCNCPoint2[8426] = {X 449.0024, Y 41.4021, Z -3.0000, A 0.000, B 0.000, C 0.000 }
gfCNCPoint2[8427] = {X 449.6384, Y 40.6660, Z -3.0000, A 0.000, B 0.000, C 0.000 }
gfCNCPoint2[8428] = {X 449.6384, Y 35.0338, Z -3.0000, A 0.000, B 0.000, C 0.000 }
gfCNCPoint2[8429] = {X 447.8159, Y 35.0338, Z -3.0000, A 0.000, B 0.000, C 0.000 }
gfCNCPoint2[8430] = {X 443.7925, Y 42.8674, Z -3.0000, A 0.000, B 0.000, C 0.000 }
gfCNCPoint2[8431] = {X 443.9302, Y 43.5100, Z -3.0000, A 0.000, B 0.000, C 0.000 }
gfCNCPoint2[8432] = {X 443.9803, Y 44.1653, Z -3.0000, A 0.000, B 0.000, C 0.000 }
gfCNCPoint2[8433] = {X 443.9805, Y 45.0000, Z -3.0000, A 0.000, B 0.000, C 0.000 }
gfCNCPoint2[8434] = {X 443.9242, Y 45.7387, Z -3.0000, A 0.000, B 0.000, C 0.000 }
gfCNCPoint2[8435] = {X 443.7568, Y 46.4603, Z -3.0000, A 0.000, B 0.000, C 0.000 }
gfCNCPoint2[8436] = {X 443.3474, Y 47.4038, Z -3.0000, A 0.000, B 0.000, C 0.000 }
gfCNCPoint2[8437] = {X 442.7493, Y 48.2405, Z -3.0000, A 0.000, B 0.000, C 0.000 }
gfCNCPoint2[8438] = {X 441.9891, Y 48.9332, Z -3.0000, A 0.000, B 0.000, C 0.000 }
gfCNCPoint2[8439] = {X 441.1006, Y 49.4513, Z -3.0000, A 0.000, B 0.000, C 0.000 }
gfCNCPoint2[8440] = {X 440.1232, Y 49.7716, Z -3.0000, A 0.000, B 0.000, C 0.000 }
gfCNCPoint2[8441] = {X 439.1005, Y 49.8800, Z -3.0000, A 0.000, B 0.000, C 0.000 }
gfCNCPoint2[8442] = {X 432.5144, Y 49.8800, Z -3.0000, A 0.000, B 0.000, C 0.000 }
gfCNCPoint2[8443] = {X 431.6014, Y 49.7938, Z -3.0000, A 0.000, B 0.000, C 0.000 }
gfCNCPoint2[8444] = {X 430.7206, Y 49.5383, Z -3.0000, A 0.000, B 0.000, C 0.000 }
gfCNCPoint2[8445] = {X 429.8343, Y 49.0782, Z -3.0000, A 0.000, B 0.000, C 0.000 }
gfCNCPoint2[8446] = {X 429.0603, Y 48.4473, Z -3.0000, A 0.000, B 0.000, C 0.000 }
gfCNCPoint2[8447] = {X 428.4309, Y 47.6720, Z -3.0000, A 0.000, B 0.000, C 0.000 }
gfCNCPoint2[8448] = {X 427.9725, Y 46.7848, Z -3.0000, A 0.000, B 0.000, C 0.000 }
gfCNCPoint2[8449] = {X 427.7197, Y 45.9083, Z -3.0000, A 0.000, B 0.000, C 0.000 }
gfCNCPoint2[8450] = {X 427.6344, Y 45.0000, Z -3.0000, A 0.000, B 0.000, C 0.000 }
gfCNCPoint2[8451] = {X 427.6344, Y 44.2089, Z -3.0000, A 0.000, B 0.000, C 0.000 }
gfCNCPoint2[8452] = {X 427.7263, Y 43.2661, Z -3.0000, A 0.000, B 0.000, C 0.000 }
gfCNCPoint2[8453] = {X 427.9987, Y 42.3588, Z -3.0000, A 0.000, B 0.000, C 0.000 }
